(* Logix 5000 project; controller LeakTestAuto vendor 1 type 14 code 226 rev 37.11; software revision 37.01; part 2 of 13 *)
(* tags used below, declared in another part *)
   PLC : AOI_PLC;

ADD_ON_INSTRUCTION AOI_RFIDCompare   (* revision 1.0, ExecuteEnableInFalse *)
VAR_IN_OUT
   ExpectedResult : SINT[5,12]; {required}
   ExpectedResultIndex : DINT; {required}
END_VAR
VAR_OUTPUT
   Match : BOOL; {access Read Only, visible}
END_VAR
VAR_IN_OUT
   ReadBuffer : SINT[8000]; {required}
END_VAR
VAR
   i : DINT; {access None}
END_VAR

ROUTINE EnableInFalse   (* structured text *)
   Match := 0;
END_ROUTINE

ROUTINE Logic   (* structured text *)
   Match := 0;
   
   FOR i := 0 TO 11 DO
       IF ReadBuffer[i] <> ExpectedResult[ExpectedResultIndex, i] THEN
           EXIT;
       END_IF;
   END_FOR;
   
   IF i = 12 THEN
       Match := 1;
   END_IF;
END_ROUTINE
END_ADD_ON_INSTRUCTION

ADD_ON_INSTRUCTION AOI_RobotPositions   (* revision 1.0 *)
VAR_OUTPUT
   LoadingNest : DINT; {access Read Only}
   Barcode : DINT; {access Read Only}
   TestingNest1 : DINT; {access Read Only}
   TestingNest2 : DINT; {access Read Only}
   PassChute : DINT; {access Read Only}
   FailChute : DINT; {access Read Only}
END_VAR

ROUTINE Logic   (* structured text *)
   LoadingNest := 0;
   Barcode := 1;
   TestingNest1 := 2;
   TestingNest2 := 3;
   PassChute := 4;
   FailChute := 5;
END_ROUTINE
END_ADD_ON_INSTRUCTION

ADD_ON_INSTRUCTION AOI_Sequencer_x64   (* revision 1.0 *)
VAR_IN_OUT
   SequenceStructure : udt_SequenceStructure_X64; {required}
END_VAR
VAR_INPUT
   inpNextStepInterlock : BOOL; {access Read Only, required}
   inpCyclePause : BOOL; {access Read Only, required}
   inpStepMode : BOOL; {access Read Only, required}
END_VAR
VAR
   FFLUDumpREAL : REAL; {access None}
   Seq_FFLU_Cycle : CONTROL := (LEN := 10); {access None}
   Seq_FFLU_Step : CONTROL := (LEN := 64); {access None}
   Seq_FFLU_StepHist : CONTROL := (LEN := 64); {access None}
   FFLUDumpINT : INT; {access None}
   AvgContol : CONTROL := (LEN := 10); {access None}
END_VAR

ROUTINE Logic   (* ladder *)
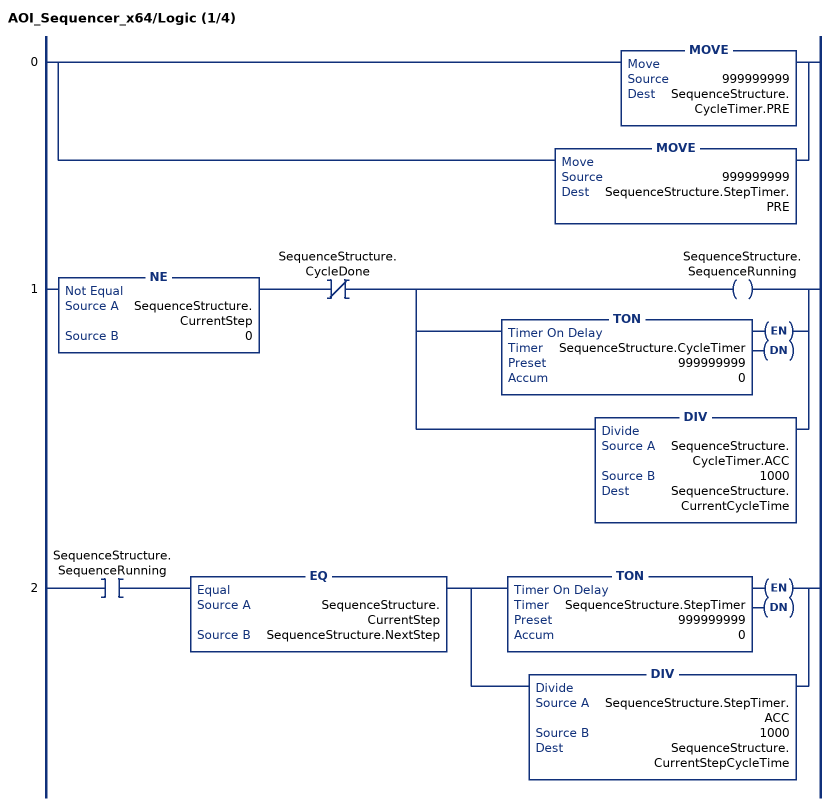
   0: [MOVE(999999999,SequenceStructure.CycleTimer.PRE) ,MOVE(999999999,SequenceStructure.StepTimer.PRE) ];
   1: NE(SequenceStructure.CurrentStep,0)XIO(SequenceStructure.CycleDone)[OTE(SequenceStructure.SequenceRunning) ,TON(SequenceStructure.CycleTimer,999999999,0) ,DIV(SequenceStructure.CycleTimer.ACC,1000,SequenceStructure.CurrentCycleTime) ];
   2: XIC(SequenceStructure.SequenceRunning)EQ(SequenceStructure.CurrentStep,SequenceStructure.NextStep)[TON(SequenceStructure.StepTimer,999999999,0) ,DIV(SequenceStructure.StepTimer.ACC,1000,SequenceStructure.CurrentStepCycleTime) ];
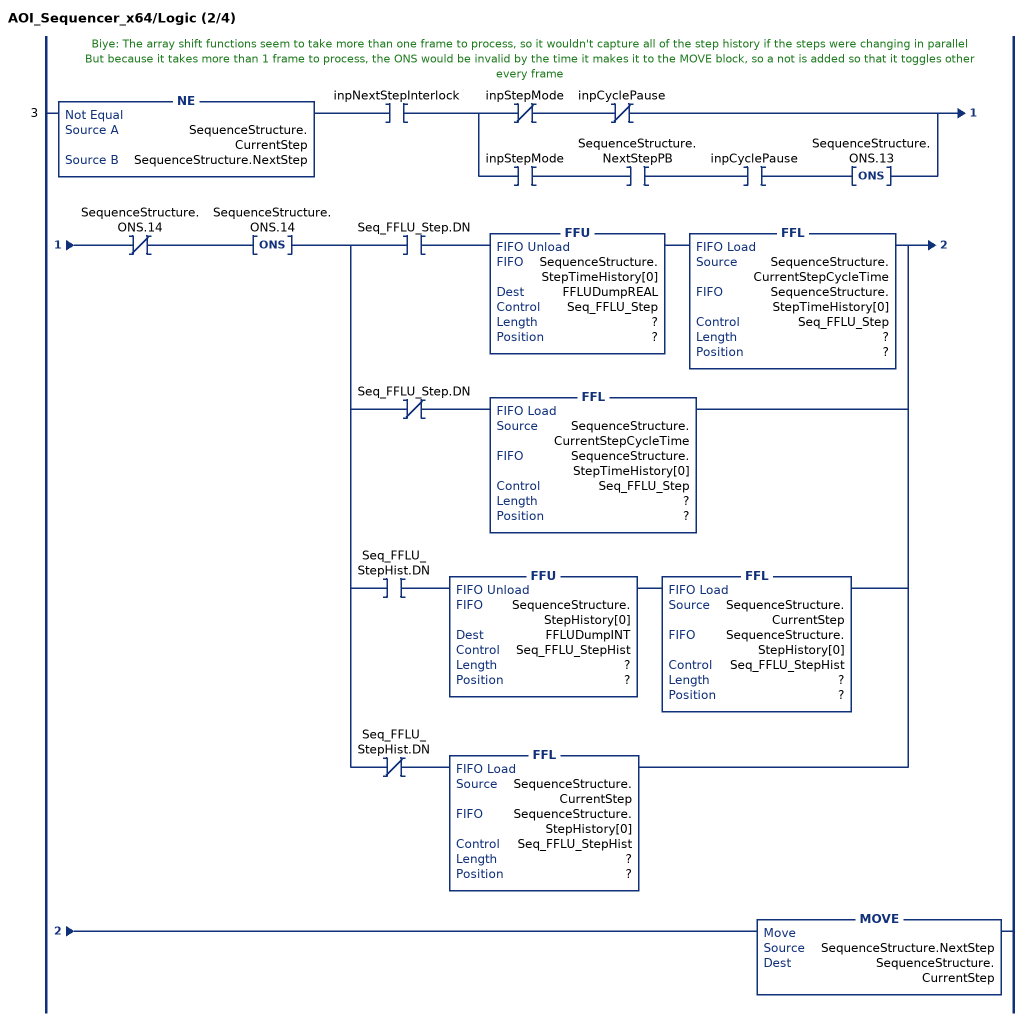
   // Biye: The array shift functions seem to take more than one frame to process, so it wouldn't capture all of the step history if the steps were changing in parallel
   // But because it takes more than 1 frame to process, the ONS would be invalid by the time it makes it to the MOVE block, so a not is added so that it toggles other every frame
   3: NE(SequenceStructure.CurrentStep,SequenceStructure.NextStep)XIC(inpNextStepInterlock)[XIO(inpStepMode) XIO(inpCyclePause) ,XIC(inpStepMode) XIC(SequenceStructure.NextStepPB) XIC(inpCyclePause) ONS(SequenceStructure.ONS.13) ]XIO(SequenceStructure.ONS.14)ONS(SequenceStructure.ONS.14)[XIC(Seq_FFLU_Step.DN) FFU(SequenceStructure.StepTimeHistory[0],FFLUDumpREAL,Seq_FFLU_Step,?,?) FFL(SequenceStructure.CurrentStepCycleTime,SequenceStructure.StepTimeHistory[0],Seq_FFLU_Step,?,?) ,XIO(Seq_FFLU_Step.DN) FFL(SequenceStructure.CurrentStepCycleTime,SequenceStructure.StepTimeHistory[0],Seq_FFLU_Step,?,?) ,XIC(Seq_FFLU_StepHist.DN) FFU(SequenceStructure.StepHistory[0],FFLUDumpINT,Seq_FFLU_StepHist,?,?) FFL(SequenceStructure.CurrentStep,SequenceStructure.StepHistory[0],Seq_FFLU_StepHist,?,?) ,XIO(Seq_FFLU_StepHist.DN) FFL(SequenceStructure.CurrentStep,SequenceStructure.StepHistory[0],Seq_FFLU_StepHist,?,?) ]MOVE(SequenceStructure.NextStep,SequenceStructure.CurrentStep);
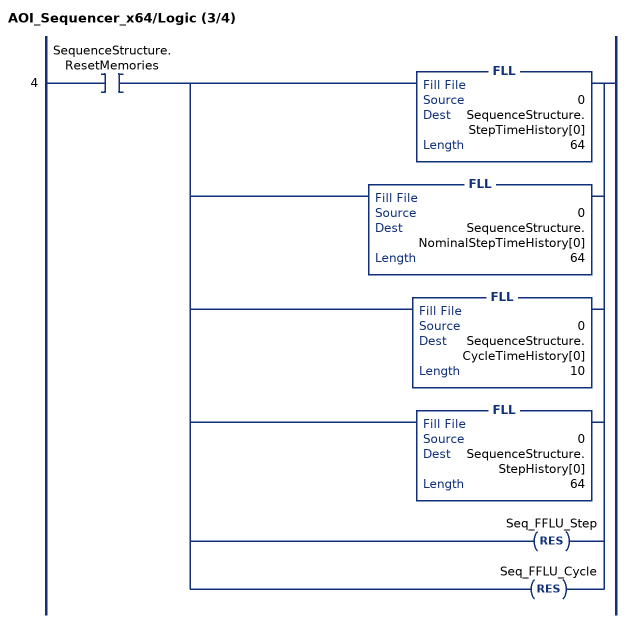
   4: XIC(SequenceStructure.ResetMemories)[FLL(0,SequenceStructure.StepTimeHistory[0],64) ,FLL(0,SequenceStructure.NominalStepTimeHistory[0],64) ,FLL(0,SequenceStructure.CycleTimeHistory[0],10) ,FLL(0,SequenceStructure.StepHistory[0],64) ,RES(Seq_FFLU_Step) ,RES(Seq_FFLU_Cycle) ];
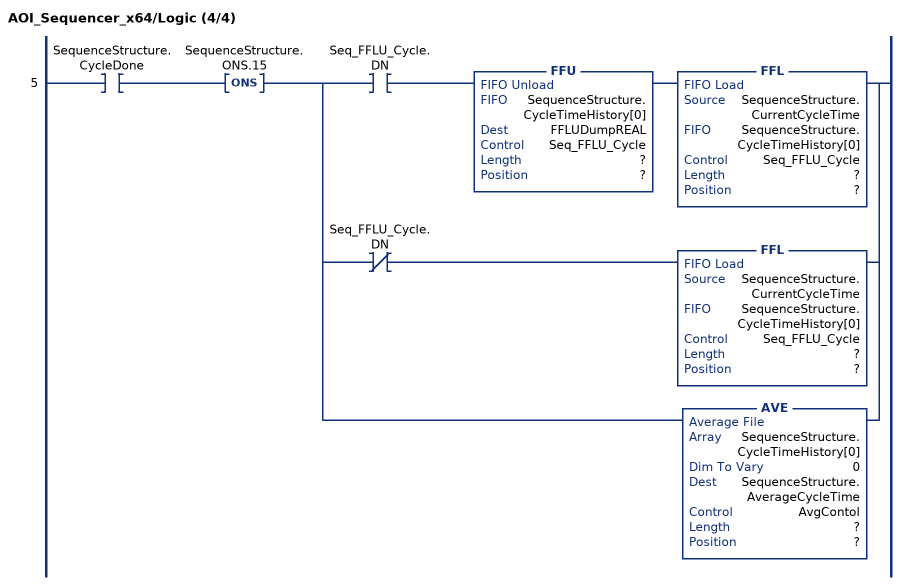
   5: XIC(SequenceStructure.CycleDone)ONS(SequenceStructure.ONS.15)[XIC(Seq_FFLU_Cycle.DN) FFU(SequenceStructure.CycleTimeHistory[0],FFLUDumpREAL,Seq_FFLU_Cycle,?,?) FFL(SequenceStructure.CurrentCycleTime,SequenceStructure.CycleTimeHistory[0],Seq_FFLU_Cycle,?,?) ,XIO(Seq_FFLU_Cycle.DN) FFL(SequenceStructure.CurrentCycleTime,SequenceStructure.CycleTimeHistory[0],Seq_FFLU_Cycle,?,?) ,AVE(SequenceStructure.CycleTimeHistory[0],0,SequenceStructure.AverageCycleTime,AvgContol,?,?) ];
END_ROUTINE
END_ADD_ON_INSTRUCTION

ADD_ON_INSTRUCTION AOI_StandardSeqSteps   (* revision 1.0 *)
VAR_OUTPUT
   Start : DINT; {access Read Only}
   ResultProcessing : DINT; {access Read Only}
   Complete : DINT; {access Read Only}
END_VAR

ROUTINE Logic   (* structured text *)
   Start := 1000;
   ResultProcessing := 8000;
   Complete := 9000;
END_ROUTINE
END_ADD_ON_INSTRUCTION

ADD_ON_INSTRUCTION INT_TO_BYTE   (* revision 1.0 *)
// It converts the INT to upper and lower nibbles
VAR_INPUT
   Input : INT;
END_VAR
VAR_OUTPUT
   OutUpperNibble : INT;
   OutLowerNibble : INT;
   iLowNib : INT; {access None}
   iUpNib : INT; {access None}
END_VAR

ROUTINE Logic   (* structured text *)
   iUpNib := Input/256;
   OutUpperNibble := iUpNib;
   iLowNib := Input -(iUpNib * 256);
   OutLowerNibble := iLowNib;
   
END_ROUTINE
END_ADD_ON_INSTRUCTION

ADD_ON_INSTRUCTION RWH_CMD   (* revision 1.1, ExecutePrescan *)
// AOI developed to handle to communicate with DTE102 , it handles 12 features of DTE 102.
// Revision note:
// Added isiModuleID, iiInputStartAdd, iiOutputStartAdd parameters for flexibility
VAR_IN_OUT
   iarsiInputFromDTE : SINT[496]; {required}   // Input array from DTE to PLC
END_VAR
VAR_INPUT
   ixConnOK : BOOL; {required}   // Connection to DTE from PLC, LIVE Status
   ixExecute : BOOL; {required}   // Rising edge : Execute selected user command.
   isiModuleID : SINT; {required}   // It indicates the module id set in the configuration to use each channel with different no of block size Please map this varible to DTE102:C.IO_x_module_identifier in controller tags. x = channel no on which RWH_CMD AOI is to be used
   iiInputStartAdd : INT; {required}   // It is the start of the DTE102:I from which the data has to be read depending upon the channel is being used by the user
   iiOutputStartAdd : INT; {required}   // It is the start of the DTE102:O to which the data has to be written depending upon the channel is being used by the user
   iiCmdCode : INT; {required}   // Command Mode for Function ID 11 and 12. For details refer user manual
   isiFunctionID : SINT; {required}   // ID of DTE10x command to be executed. For details refer user manual
   iiRdWrLength : INT; {required}   // data length (in BYTEs) to read/write USER memory on tag
   iiRdWrStartAddr : INT; {required}   // start address to read/write USER memory on tag
END_VAR
VAR_IN_OUT
   iarsiSendBuf : SINT[8000]; {required}   // send buffer for data to write to USER memory on tag
END_VAR
VAR_OUTPUT
   oxBusy : BOOL; {access Read Only, visible}   // Function block is busy, no new command possible
   oxDone : BOOL; {access Read Only, visible}   // TRUE: Operation resulted in error
   oxError : BOOL; {access Read Only, visible}   // TRUE: Operation resulted in error
   odiStatus : DINT; {access Read Only, visible}   // Status information or error code. For details refer user manual
   oxTagPresent : BOOL; {access Read Only, visible}   // TRUE : Tag present in field, FALSE : Tag not in field
   oiRcvdLength : INT; {access Read Only, visible}   // data length (in BYTEs) read from the tag
END_VAR
VAR_IN_OUT
   oarsiRcvBuf : SINT[8000]; {required}   // receive buffer for data from tag
END_VAR
VAR_OUTPUT
   oiDiagLength : INT; {access Read Only, visible}   // number of diagnostic data erros
END_VAR
VAR_IN_OUT
   oardiDiagData : DINT[4]; {required}   // Array with diagonostic data
   oarsiOutputToDTE : SINT[496]; {required}   // Output array from PLC to DTE
END_VAR
VAR
   iRcvdLength : INT;   // Local tag - calculates the received data length from PLC
   iLoopHandlerVar2 : INT;   // Local tag - Loop Handler variable 2
   iLoopHandlerVar1 : INT;   // Local tag - Loop Handler variable 1
   iActSizeOfSendBuf : INT;   // Local tag - Calculates the actual array size of the input array
   iActSizeOfRcvBuf : INT;   // Local tag - Calculates the actual array size of the recieve data array
   iActSizeOfOutputToDTE : INT;   // Local tag - Calculates the actual array size of the output array
   iActSizeOfInputFromDTE : INT;   // Local tag - Calculates the actual array size of the input array
   iBufferOffset : INT;   // Local tag - calculates the start adddress to read/write the data in buffer in case of ,ultiple cycles
   siActiveFunctionID : SINT;   // Loca tag - Latch the value of the selected ID to generate the error if t changes while function block is busy.
   siActiveModuleID : SINT; {access None}   // Local tag - indicates the active module id selected by user
   ciStateMachineSeparator : INT; {access None}   // Local tag = constant value of 1000. It separates the steps in state machine as per Function ID.
   iCmdCode : INT; {access None}   // Loca tag - Latch the value of the selected Cmd Code to generate the error if it changes while function block is busy.
   iLowerLimitInputStartAdd : INT; {access None}   // Local tag for limit the start address of input
   iUpperLimitInputStopAdderess : INT; {access None}   // Local tag - limit the upper range of input stop address
   iLowerLimitOutputStartAdd : INT; {access None}   // Local tag for limit the start address of output
   iUpperLimitOutputStopAdderess : INT; {access None}   // Local tag - limit the upper range of output stop address
   iActiveInputStartAdd : INT; {access None}   // Local Tag - Indicates the active input start adderess
   iActiveOutputStartAdd : INT; {access None}   // Local tag - Indicates the active output start address
   iArraySize : INT; {access None}
   iLengthToReadWriteInLastCycle : INT;   // Local tag to clculate the no of data byte to read/write in last cycle
   iNoCyclesReqToReadWriteCompleteData : INT;   // Local tag - Calculates the no of cycles required to read/write the data to/from DTE.
   iSingleCycleDataExchangeLimitInBytes : INT; {access None}   // Local tag - Decides the limit for bytes to exchange in one PLC cycle
   iTotalRcvdLength : INT; {access Read Only}   // data length (in BYTEs) read from the tag
   fb_OSRI_Execute : FBD_ONESHOT; {access None}   // Local tag - Detects the rising edge of the execute trigger. Avoids the multiple triggers for single command
   fb_DataAddress : INT_TO_BYTE; {access None}
   ardiDiagData : DINT[4]; {access None}   // Local tag -Array with diagonostic data
   xMultipleCyclesReq : BOOL;   // Local tag - Status for single or multiple cycle requirement to read / write data. if xMultipleCyclesReq = 0 then data transmission takes one cycle else it takes >1 cycles.
   fb_CmdCode : INT_TO_BYTE; {access None}   // Local tag = function block to convert cmd code to MSB and LSB.
   fb_OSRI_TagPresent : FBD_ONESHOT; {access None}   // Local tag = checks for tag present rising edge to read / write asynchronous commands
   fb_DataLength : INT_TO_BYTE; {access None}
   fb_SINT_TO_INT : SINT_TO_INT; {access None}
   scDTE102_Handling : DTE102_CmdModule; {access None}
   iStateMachine_RWH_CMD : INT;   // Local tag - State machine handling variable for AOI logic
END_VAR

ROUTINE Logic   (* structured text *)
   (*// ******************************************************************************************************
   // Disclaimer OF Warranties
   (*
   	ifm disclaims to the fullest extent authorized by law any and all warranties,
   	whether express or implied, including, without limitation,
   	any implied warranties of title, non-infringement, quiet enjoyment,
   	integration, merchantability or fitness for a particular purpose.
   
   	Without limitation of the foregoing, ifm expressly does not warrant that:
   	(a)  the software will meet your requirements or expectations;
   	(b)  the software or the software content will be free of bugs, errors,
   			 viruses or other defects;
   	(c)  any results, output, or data provided through or generated by the software
   			 will be accurate, up-to-date, complete or reliable;
   	(d)  the software will be compatible with third party software;
   	(e)  any errors in the software will be corrected
   
   
   	DEMO SOFTWARE AND TEMPLATES
   
   	Demo software and templates are provided “as is” and “as available”,
   	without any warranty of any kind, either express or implied.
   	The User acknowledges and agrees to use the software at User’s own risk.
   	In no event shall ifm be held liable for any direct, indirect, incidental
   	or consequential damages arising out of the use of or inability to use the software.
   	User may use the software solely for demonstration purposes
   	and to assess the software functionalities and capabilities.
   
   
   	Software written specifically for Customer
   
   	1. The software created and used is put together by ifm specially to the customer
   		 using modular software components made by ifm for numerous applications (Standard software modules)
   		 and adapted to the contractual service required (customer-specific application program).
   
   	2. Upon complete payment of the purchase price for the customer-specific application program,
   		 ifm transfers the non-exclusive, locally and temporarily unrestricted usage right
   		 thereof to the customer, without the customer acquiring any rights of any kind
   		 to the standard software module on which the individual or customer-specific adaptation is based.
   		 Notwithstanding these provisions, ifm reserves the right to produce and offer
   		 customer specific software solutions of the same kind for other customers
   		 based on other terms of reference. In any case ifm retains a simple right of usage
   		 of the customer–specific solution for internal purposes.
   
   	3. Upon acceptance of the program, User acknowledges and agrees to use the software
   		 at User’s own risk. User also acknowledges and agrees upon acceptance of the program
   		 that the software meets the requirements of the specifications agreed upon.
   		 ifm disclaims any and all warranties, in particular regarding fitness of the software
   		 for a particular purpose.
   ******************************************************************************************************
   *)
   (* Revision history:
   3rd June 2022:
   New Chnage requests:
   1. check if the "get diagdata" command is send if TP bit is high and no command active
      DiagData before sending a command --> get Diagnostic shall be send automatically before executing a user command.
   
   
   24th Dec 2020:
   Fixed bug:
   	Whenever customer tries to read (one time) from offset=10, length = 10 bytes, the data is read from offset=0
   	Same for writing (one time) and write verifed (one time) operations too.
   
   26th July 2019:
   	Till now, it was assumed that after diagnostic read, maximum number of reported errors could be 4 only.
   	But, actually errors are to be read, until DIAG bit is active.
   	Fixed this in the code.
   
   19th July 2019:
   	Added following check.
   	When a execute trigger is given, and already some operation is in progress (TA <> TR).
   	Now, we wait for ongoing operation to complete.
   
   17th July 2019:
   	i. Write-verified operation: Added extra check, that the number of recieved bytes should be same as requested "iiRdWrLength"
   	ii. Added a logic to report error, in case device reports error and provides no error codes.
   
   16th July 2019:
   	i. Fixed following bugs:
   	All 4 channels were used, and given a command of "write verified" one time.
   	For every alternate channel, operation resulted in error.
   	Reason: While waiting for user action, the TR bit was not maintained same as TA
   
   9th July 2019
   	Fixed following bugs:
   	i. Parallel usage of all 4 channels, with configuration 17,17,17,14 was buggy.
   	Reason: Every fb instance's trigger reset, was overwritting DTE fieldbus output array.
   
   	ii. Write verfied was not working for channel, with module id 12. RdWrLength = 8000 bytes
   	Reason: The number of bytes to be written in last cyle, was not calculated correctly.
   *)
   (*
   Status codes:
   	0x0000 	Function completed without error.
   	0x1000	Waiting for ixConnOk = TRUE, input parameter
   	0x7000	Wait for start of command
   	0x7001	Wait for Rising edge of the TP Bit in case of asynchronous commands
   	0x7102	Read the USER Memory
   	0x7103	Complete reading of the USER Memory
   	0x7202	Write to the USER Memory
   	0x7203	Complete writing to the USER Memory
   	0x7302	Read UID
   	0x7303	Complete reading UID
   	0x7402	Read Diagnostic data
   	0x7403	Complete reading the Diagnostic data
   	0x7501	Antenna OFF command
   	0x7502	Complete Antenna OFF command
   	0x7601	Antenna ON command
   	0x7602	Complete Antenna ON command
   	0x7701	Read device parameters one time Command
   	0x7702	Complete read device parameters one time command
   	0x7801	Set device parameters one time Command
   	0x7802	Complete Set device parameters one time command
   
   Error codes:
   	0x8000 	Evaluation unit indicates an error; evaluate the diagnostic data in the oardiDiagData output parameter. For the error codes see the device manual
   	0x8101 	isiFunctionID input parameter invalid
   
   	0x8104	Different sizes of the iarsiInputFromDTE input parameter and oarsiOutputToDTE output parameter
   	0x8107	iiCmdCode = Invalid, but selected ID is 11 or 12
   	0x8109	iiRdWrStartAddr input is invalid
   	0x8110	Antenna already OFF.
   	0x8111	Antenna already ON.
   	0x8112	Wrong Module ID entered by user
   	0x8113	Wrong Input Start Address entered by user
   	0x8114	Wrong Output Start Address entered by user
   	0x8201	ixConnOk input parameter = FALSE during command execution.
   	0x8301	Start of a command while the function block is busy (oxBusy = TRUE)
   	0x8302	Start of a command with antenna switched off.
   	0x8303	Function ID changed while function block is BUSY.
   	0x8304	Start of a command without tag in the antenna field
   	0x8305	iiRdWrLength input parameter <= 0 or greater than the defined receive buffer (oarsiRcvBuf)
   	0x8306	iiRdWrLength input parameter <= 0 or greater than the defined send buffer (iarsiSendBuf)
   	0x8307	Invalid Read Write data length if asynchronous command is selected
   	0x8308	Command Code changed while function block is BUSY.
   	0x8309	Module ID changed when function block is BUSY
   	0x8310	Input start address changed when function block is BUSY
   	0x8311	Output start address changed when function block is BUSY
   	0x8313 	Write-verified: Complete data could not be written
   	0x8314  Device reported error, but provided no diagonostic codes
    	0x8315	Read data: Complete data could not be read
   	0x8316	Write data: Complete data could not be written
   *)
   	// Execute Trigger
   	fb_OSRI_Execute.InputBit := ixExecute;
   	OSRI(fb_OSRI_Execute);
   
   	// If function block is busy and following conditions occure then go to error state
   	// 1. Connection Lost
   	// 2. Multiple Execute Triggers
   	// 3. ID Change by user
   	// 4. Command code changed by the user
   	// 5. Module ID changed by the user
   	// 6. Input start add changed by the user
   	// 7. Output start add changed by the user
   
   	IF(iStateMachine_RWH_CMD > 0 AND iStateMachine_RWH_CMD < 20000)THEN
   		IF(NOT(ixConnOK))THEN							// No Connection to DTE
   			oxBusy := 1;
   			oxDone := 0;
   			oxError := 0;
   			odiStatus := 16#8201; //ixConnOk input parameter = FALSE during command execution.
   			iStateMachine_RWH_CMD := 20000;
   		ELSIF(fb_OSRI_Execute.OutputBit)THEN			// Multiple Execute Triggers
   			oxBusy := 1;
   			oxDone := 0;
   			oxError := 0;
   			odiStatus := 16#8301; //Start of a command while the function block is busy (oxBusy = TRUE)
   			iStateMachine_RWH_CMD := 20000;
   		ELSIF(isiFunctionID<>siActiveFunctionID)THEN	// Function ID Changed by user when function is Active
   			oxBusy := 1;
   			oxDone := 0;
   			oxError := 0;
   			odiStatus := 16#8303; //Function ID changed while function block is BUSY.
   			iStateMachine_RWH_CMD := 20000;
   		ELSIF(iiCmdCode <> iCmdCode)THEN				// Command code changed by user when function is Active
   			oxBusy := 1;
   			oxDone := 0;
   			oxError := 0;
   			odiStatus := 16#8308; //Command Code changed while function block is BUSY.
   			iStateMachine_RWH_CMD := 20000;
   		ELSIF(siActiveModuleID <> isiModuleID)THEN
   			oxBusy := 1;
   			oxDone := 0;
   			oxError := 0;
   			odiStatus := 16#8309; 						// Module ID changed by user when function is Active
   			iStateMachine_RWH_CMD := 20000;
   		ELSIF(iActiveInputStartAdd <> iiInputStartAdd)THEN
   			oxBusy := 1;
   			oxDone := 0;
   			oxError := 0;
   			odiStatus := 16#8310; 						// Input Start Address changed by user when function is Active
   			iStateMachine_RWH_CMD := 20000;
   		ELSIF(iActiveOutputStartAdd <> iiOutputStartAdd)THEN
   			oxBusy := 1;
   			oxDone := 0;
   			oxError := 0;
   			odiStatus := 16#8311; 						// Output Start Address changed by user when function is Active
   			iStateMachine_RWH_CMD := 20000;
   		END_IF;
   	END_IF;
   
   	IF(iiInputStartAdd >= 0 AND iiInputStartAdd < 496)AND(iiOutputStartAdd >= 0 AND iiOutputStartAdd < 496)THEN
   		// Maping of Input bits
   		scDTE102_Handling.Status.TP		:=	iarsiInputFromDTE[iiInputStartAdd].0;
   		scDTE102_Handling.Status.AI 	:=	iarsiInputFromDTE[iiInputStartAdd].1;
   		scDTE102_Handling.Status.WA 	:=	iarsiInputFromDTE[iiInputStartAdd].2;
   		scDTE102_Handling.Status.RA 	:=	iarsiInputFromDTE[iiInputStartAdd].3;
   		scDTE102_Handling.Status.UA 	:=	iarsiInputFromDTE[iiInputStartAdd].4;
   		scDTE102_Handling.Status.EA 	:=	iarsiInputFromDTE[iiInputStartAdd].5;
   		scDTE102_Handling.Status.DA 	:=	iarsiInputFromDTE[iiInputStartAdd].6;
   		scDTE102_Handling.Status.DIAG	:=	iarsiInputFromDTE[iiInputStartAdd].7;
   
   
   		scDTE102_Handling.Status.TA						:=	iarsiInputFromDTE[iiInputStartAdd+1].0;
   		iarsiInputFromDTE[iiInputStartAdd+1].1			:=	iarsiInputFromDTE[iiInputStartAdd+1].1;
   		iarsiInputFromDTE[iiInputStartAdd+1].2 			:=	iarsiInputFromDTE[iiInputStartAdd+1].2;
   		iarsiInputFromDTE[iiInputStartAdd+1].3 			:=	iarsiInputFromDTE[iiInputStartAdd+1].3;
   		iarsiInputFromDTE[iiInputStartAdd+1].4 			:=	iarsiInputFromDTE[iiInputStartAdd+1].4;
   		iarsiInputFromDTE[iiInputStartAdd+1].5 			:=	iarsiInputFromDTE[iiInputStartAdd+1].5;
   		iarsiInputFromDTE[iiInputStartAdd+1].6 			:=	iarsiInputFromDTE[iiInputStartAdd+1].6;
   		scDTE102_Handling.Status.CA 					:=	iarsiInputFromDTE[iiInputStartAdd+1].7;
   	END_IF;
   
   	// Mapping tag Present bit to output variable
   	oxTagPresent := scDTE102_Handling.Status.TP;
   
   	// Asynchronous commands :- Check For tag Present bit
   	fb_OSRI_TagPresent.InputBit := scDTE102_Handling.Status.TP;
   	OSRI(fb_OSRI_TagPresent);
   
   
   CASE iStateMachine_RWH_CMD OF
   	/// This case checks the inputs entered by user properly or not.
   	0:
   		scDTE102_Handling.ActivateCommand.TR	:= (iarsiInputFromDTE[iiInputStartAdd+1].0); //Do not accidently trigger a command
   
   		// getting the sizes of arrays used in function block to check correct sizes declared by user.
   		SIZE(iarsiInputFromDTE,0,iActSizeOfInputFromDTE);
   		SIZE(oarsiOutputToDTE,0,iActSizeOfOutputToDTE);
   		SIZE(iarsiSendBuf,0,iActSizeOfSendBuf);
   		SIZE(oarsiRcvBuf,0,iActSizeOfRcvBuf);
   
   		// Logic to identify the module ID and related Data buffer size required for operations and start address for reading and writting
   		CASE isiModuleID OF
   			12 :
   				iLowerLimitInputStartAdd := 0;
   				iUpperLimitInputStopAdderess := iActSizeOfInputFromDTE - 26;
   				iLowerLimitOutputStartAdd := 0;
   				iUpperLimitOutputStopAdderess := iActSizeOfOutputToDTE - 26;
   				iSingleCycleDataExchangeLimitInBytes := 20;
   			13 :
   				iLowerLimitInputStartAdd := 0;
   				iUpperLimitInputStopAdderess := iActSizeOfInputFromDTE - 46;
   				iLowerLimitOutputStartAdd := 0;
   				iUpperLimitOutputStopAdderess := iActSizeOfOutputToDTE - 46;
   				iSingleCycleDataExchangeLimitInBytes := 40;
   			14 :
   				iLowerLimitInputStartAdd := 0;
   				iUpperLimitInputStopAdderess := iActSizeOfInputFromDTE - 66;
   				iLowerLimitOutputStartAdd := 0;
   				iUpperLimitOutputStopAdderess := iActSizeOfOutputToDTE - 66;
   				iSingleCycleDataExchangeLimitInBytes := 60;
   			15 :
   				iLowerLimitInputStartAdd := 0;
   				iUpperLimitInputStopAdderess := iActSizeOfInputFromDTE - 86;
   				iLowerLimitOutputStartAdd := 0;
   				iUpperLimitOutputStopAdderess := iActSizeOfOutputToDTE - 86;
   				iSingleCycleDataExchangeLimitInBytes := 80;
   			16 :
   				iLowerLimitInputStartAdd := 0;
   				iUpperLimitInputStopAdderess := iActSizeOfInputFromDTE - 106;
   				iLowerLimitOutputStartAdd := 0;
   				iUpperLimitOutputStopAdderess := iActSizeOfOutputToDTE - 106;
   				iSingleCycleDataExchangeLimitInBytes := 100;
   			17 :
   				iLowerLimitInputStartAdd := 0;
   				iUpperLimitInputStopAdderess := iActSizeOfInputFromDTE - 126;
   				iLowerLimitOutputStartAdd := 0;
   				iUpperLimitOutputStopAdderess := iActSizeOfOutputToDTE - 126;
   				iSingleCycleDataExchangeLimitInBytes := 120;
   			18 :
   				iLowerLimitInputStartAdd := 0;
   				iUpperLimitInputStopAdderess := iActSizeOfInputFromDTE - 146;
   				iLowerLimitOutputStartAdd := 0;
   				iUpperLimitOutputStopAdderess := iActSizeOfOutputToDTE - 146;
   				iSingleCycleDataExchangeLimitInBytes := 140;
   			19 :
   				iLowerLimitInputStartAdd := 0;
   				iUpperLimitInputStopAdderess := iActSizeOfInputFromDTE - 166;
   				iLowerLimitOutputStartAdd := 0;
   				iUpperLimitOutputStopAdderess := iActSizeOfOutputToDTE - 166;
   				iSingleCycleDataExchangeLimitInBytes := 160;
   		END_CASE;
   
   		// Checking all input parameters
   		IF(fb_OSRI_Execute.OutputBit)THEN //Received trigger
   			oxBusy := 1;
   			oxDone := 0;
   			oxError := 0;
   			IF(NOT(ixConnOK))THEN
   				odiStatus := 16#8201;					// ixConnOk input parameter = FALSE during command execution.
   				iStateMachine_RWH_CMD := 20000;
   			ELSIF(isiModuleID < 12 OR isiModuleID > 19)THEN
   				odiStatus := 16#8112;					// Wrong Module ID entered by user.
   				iStateMachine_RWH_CMD := 20000;
   			ELSIF(iiInputStartAdd < iLowerLimitInputStartAdd OR iiInputStartAdd > iUpperLimitInputStopAdderess)THEN
   				odiStatus := 16#8113;					// Wrong Input Start Address entered by user.
   				iStateMachine_RWH_CMD := 20000;
   			ELSIF(iiOutputStartAdd < iLowerLimitOutputStartAdd OR iiOutputStartAdd > iUpperLimitOutputStopAdderess)THEN
   				odiStatus := 16#8114;					// Wrong Output Start Address entered by user.
   				iStateMachine_RWH_CMD := 20000;
   			ELSIF(isiFunctionID < 1 OR isiFunctionID > 12)THEN
   				odiStatus := 16#8101;					// isiFunctionID input parameter invalid
   				iStateMachine_RWH_CMD := 20000;
   			ELSIF((isiFunctionID = 11 AND(iiCmdCode<>25288 AND iiCmdCode<>25289 AND (iiCmdCode < 25293 OR iiCmdCode > 25299))) OR
   			  	 (isiFunctionID = 12 AND (iiCmdCode< 26070 OR iiCmdCode > 26077)))THEN
   				odiStatus := 16#8107;					// iiCmdCode = Invalid, but selected ID is 11 or 12
   				iStateMachine_RWH_CMD := 20000;
   			ELSIF(iActSizeOfInputFromDTE <> iActSizeOfOutputToDTE)THEN
   				odiStatus := 16#8104;					// Different sizes of the iarsiInputFromDTE input parameter and oarsiOutputToDTE output parameter
   				iStateMachine_RWH_CMD := 20000;
   			ELSIF((iiRdWrLength < 1 or iiRdWrLength > iActSizeOfRcvBuf)AND(isiFunctionID <> 9 AND isiFunctionID <> 10 AND isiFunctionID <> 1 AND isiFunctionID <> 2 AND isiFunctionID <> 11 AND isiFunctionID <> 12)) OR
   				 ((iiRdWrLength < 1 or iiRdWrLength > iActSizeOfRcvBuf) AND((isiFunctionID = 11 AND iiCmdCode = 16#62D1)OR(isiFunctionID = 12 AND iiCmdCode = 16#65D8)))THEN
   				odiStatus := 16#8305;					// iiRdWrLength input parameter <= 0 or greater than the defined receive buffer (oarsiRcvBuf)
   				iStateMachine_RWH_CMD := 20000;
   			ELSIF((iiRdWrLength < 1 or iiRdWrLength > iActSizeOfSendBuf)AND(isiFunctionID <> 9 AND isiFunctionID <> 10 AND isiFunctionID <> 1 AND isiFunctionID <> 2 AND isiFunctionID <> 11 AND isiFunctionID <> 12)) OR
   				 ((iiRdWrLength < 1 or iiRdWrLength > iActSizeOfSendBuf) AND((isiFunctionID = 11 AND iiCmdCode = 16#62D1)OR(isiFunctionID = 12 AND iiCmdCode = 16#65D8)))THEN
   				odiStatus := 16#8306;					// iiRdWrLength input parameter <= 0 or greater than the defined send buffer (iarsiSendBuf)
   				iStateMachine_RWH_CMD := 20000;
   			ELSIF(iiRdWrLength < 1 or iiRdWrLength > (iSingleCycleDataExchangeLimitInBytes))AND((isiFunctionID = 3)OR(isiFunctionID = 5)OR(isiFunctionID = 7))THEN
   				odiStatus := 16#8307;					// Invalid Read Write data length if asynchronous command is selected.
   				iStateMachine_RWH_CMD := 20000;
   			ELSIF(scDTE102_Handling.Status.AI)AND(isiFunctionID <> 9)AND(isiFunctionID <> 10)THEN
   				odiStatus := 16#8302;					// Start of a command with antenna switched off.
   				iStateMachine_RWH_CMD := 20000;
   			ELSIF(NOT(oxTagPresent))AND(isiFunctionID <> 9)AND(isiFunctionID <> 10)AND(isiFunctionID <> 3)AND(isiFunctionID <> 5)AND(isiFunctionID <> 7)AND(isiFunctionID <> 1)THEN
   				odiStatus := 16#8304;					// Start of a command without tag in the antenna field
   				iStateMachine_RWH_CMD := 20000;
   			ELSIF((iiRdWrStartAddr < 0 OR iiRdWrStartAddr > (iActSizeOfSendBuf-iiRdWrLength))AND(isiFunctionID <> 9 AND isiFunctionID <> 10 AND isiFunctionID <> 1 AND isiFunctionID <> 2 AND isiFunctionID <> 11 AND isiFunctionID <> 12)) OR
   				 ((iiRdWrStartAddr < 0 OR iiRdWrStartAddr > (iActSizeOfSendBuf-iiRdWrLength)) AND((isiFunctionID = 11 AND iiCmdCode = 16#62D1)OR(isiFunctionID = 12 AND iiCmdCode = 16#65D8)))THEN
   				odiStatus := 16#8109;					// iiRdWrStartAddr input is invalid
   				iStateMachine_RWH_CMD := 20000;
   			ELSIF(isiFunctionID = 9)AND(scDTE102_Handling.Status.AI)THEN
   				odiStatus := 16#8110;					// Antenna already OFF.
   				iStateMachine_RWH_CMD := 20000;
   			ELSIF(isiFunctionID = 10)AND(NOT(scDTE102_Handling.Status.AI))THEN
   				odiStatus := 16#8111;					// Antenna already ON.
   				iStateMachine_RWH_CMD := 20000;
   			ELSE
   				siActiveFunctionID := isiFunctionID;	// All input parameters are valid. Start executing the selected ID.
   				iCmdCode := iiCmdCode;
   				ciStateMachineSeparator := 1000;		//cStateMachineSeparator := 1000;
   				siActiveModuleID := isiModuleID;
   				iActiveInputStartAdd := iiInputStartAdd;
   				iActiveOutputStartAdd := iiOutputStartAdd;
   				iStateMachine_RWH_CMD := 7110;
   
   			END_IF;
   		ELSE //no trigger recieved yet
   			IF(NOT(ixConnOK))THEN
   				oxBusy := 0;
   				oxDone := 0;
   				oxError := 0;
   				odiStatus := 16#1000;					//No connection to DTE.
   				iStateMachine_RWH_CMD := 0;
   			ELSE
   				oxBusy := 0;
   				oxDone := 0;
   				oxError := 0;
   				odiStatus := 16#7000;					// Connection OK, Waiting for Command.
   				iStateMachine_RWH_CMD := 0;
   			END_IF;
   		END_IF;
   
   // Get automatically existing diagnostic data before executing new user command.
   
   	7110:
   		IF(scDTE102_Handling.Status.DIAG)THEN		//  Existing Error is present
   			oxBusy := 1;
   			oxDone := 0;
   			oxError := 0;
   			scDTE102_Handling.ActivateCommand.AO	:= 0;
   			scDTE102_Handling.ActivateCommand.WR	:= 0;
   			scDTE102_Handling.ActivateCommand.RD	:= 0;
   			scDTE102_Handling.ActivateCommand.UR	:= 0;
   			scDTE102_Handling.ActivateCommand.ER	:= 0;
   			scDTE102_Handling.ActivateCommand.DR	:= 1;
   			scDTE102_Handling.ActivateCommand.CM	:= 0;
   			scDTE102_Handling.ActivateCommand.TR	:= NOT(scDTE102_Handling.Status.TA);
   			odiStatus := 16#7402;
   			iStateMachine_RWH_CMD					:= 7111;
   		ELSIF NOT(scDTE102_Handling.Status.TA XOR scDTE102_Handling.ActivateCommand.TR)THEN // Proceed,when TA=TR
   			iStateMachine_RWH_CMD := siActiveFunctionID * ciStateMachineSeparator;
   		END_IF;
   
   	7111:// waiting for fieldbus to free
   		IF NOT(scDTE102_Handling.Status.TA XOR scDTE102_Handling.ActivateCommand.TR)THEN // Proceed,when TA=TR
   			iStateMachine_RWH_CMD					:= 7112;
   		end_if;
   
   	7112:
   		IF (scDTE102_Handling.Status.DIAG)THEN		//   IF Error is present
   			oxBusy := 1;
   			oxDone := 0;
   			oxError := 0;
   			scDTE102_Handling.ActivateCommand.AO	:= 0;
   			scDTE102_Handling.ActivateCommand.WR	:= 0;
   			scDTE102_Handling.ActivateCommand.RD	:= 0;
   			scDTE102_Handling.ActivateCommand.UR	:= 0;
   			scDTE102_Handling.ActivateCommand.ER	:= 0;
   			scDTE102_Handling.ActivateCommand.DR	:= 1;
   			scDTE102_Handling.ActivateCommand.CM	:= 0;
   			scDTE102_Handling.ActivateCommand.TR	:= NOT(scDTE102_Handling.Status.TA);
   			odiStatus := 16#7402;
   			iStateMachine_RWH_CMD					:= 19000;
   		ELSIF NOT(scDTE102_Handling.Status.TA XOR scDTE102_Handling.ActivateCommand.TR)THEN // Proceed,when TA=TR
   			iStateMachine_RWH_CMD := siActiveFunctionID * ciStateMachineSeparator;
   		END_IF;
   
   	// Function ID 1 :- read the UID of the ID-tag continuously
   	1000:
   		// frame a command and send to the DTE.
   		scDTE102_Handling.ActivateCommand.AO	:= 0;
   		scDTE102_Handling.ActivateCommand.WR	:= 0;
   		scDTE102_Handling.ActivateCommand.RD	:= 0;
   		scDTE102_Handling.ActivateCommand.UR	:= 0;
   		scDTE102_Handling.ActivateCommand.ER	:= 0;
   		scDTE102_Handling.ActivateCommand.DR	:= 0;
   		scDTE102_Handling.ActivateCommand.CM	:= 0;
   		oarsiOutputToDTE[iiOutputStartAdd+2]	:= 0;
   		oarsiOutputToDTE[iiOutputStartAdd+3]	:= 0;
   		oarsiOutputToDTE[iiOutputStartAdd+4]	:= 0;
   		oarsiOutputToDTE[iiOutputStartAdd+5]	:= 0;
   		scDTE102_Handling.ActivateCommand.TR	:= NOT(scDTE102_Handling.Status.TA);
   		odiStatus := 16#7302;
   		iStateMachine_RWH_CMD					:= 1050;
   
   
   	1050:
   		IF(scDTE102_Handling.Status.DIAG)THEN		// Error in receiving  the data from DTE.
   			oxBusy := 1;
   			oxDone := 0;
   			oxError := 0;
   			scDTE102_Handling.ActivateCommand.AO	:= 0;
   			scDTE102_Handling.ActivateCommand.WR	:= 0;
   			scDTE102_Handling.ActivateCommand.RD	:= 0;
   			scDTE102_Handling.ActivateCommand.UR	:= 0;
   			scDTE102_Handling.ActivateCommand.ER	:= 0;
   			scDTE102_Handling.ActivateCommand.DR	:= 1;
   			scDTE102_Handling.ActivateCommand.CM	:= 0;
   			oarsiOutputToDTE[iiOutputStartAdd+2]	:= 16#00;
   			scDTE102_Handling.ActivateCommand.TR	:= NOT(scDTE102_Handling.Status.TA);
   			odiStatus := 16#7402;
   			iStateMachine_RWH_CMD					:= 19000;
   		ELSE										// ElSE condition, no error then read the status from the DTE.
   			IF(NOT(scDTE102_Handling.Status.TA XOR scDTE102_Handling.ActivateCommand.TR))THEN // Proceed,when TA=TR
   				SINT_TO_INT(fb_SINT_TO_INT,iarsiInputFromDTE[iiInputStartAdd+3]);
   				iRcvdLength := fb_SINT_TO_INT.oINT_var;
   				IF(iRcvdLength <> 0)THEN //Data read is non zero
   					oiRcvdLength := (iRcvdLength-2);			// Subtract 2 from actual length which is RSSI length.
   					CPS(iarsiInputFromDTE[iiInputStartAdd+6],oarsiRcvBuf[0],oiRcvdLength);
   					odiStatus := 16#7303;
   					iStateMachine_RWH_CMD := 13000;
   				ELSIF(NOT(scDTE102_Handling.Status.TP))THEN
   					oxBusy := 1;
   					oxDone := 0;
   					oxError := 0;
   					odiStatus := 16#7001;
   					iStateMachine_RWH_CMD := 1050;
   				END_IF;
   			END_IF;
   		END_IF;
   
   	// Function ID 2 :- read the UID of the ID-tag one time
   	2000:
   		// frame a command and send to the DTE.
   		scDTE102_Handling.ActivateCommand.AO	:= 0;
   		scDTE102_Handling.ActivateCommand.WR	:= 0;
   		scDTE102_Handling.ActivateCommand.RD	:= 1;
   		scDTE102_Handling.ActivateCommand.UR	:= 0;
   		scDTE102_Handling.ActivateCommand.ER	:= 0;
   		scDTE102_Handling.ActivateCommand.DR	:= 0;
   		scDTE102_Handling.ActivateCommand.CM	:= 1;
   		oarsiOutputToDTE[iiOutputStartAdd+2]	:= 0;
   		oarsiOutputToDTE[iiOutputStartAdd+3]	:= 16#02;
   		oarsiOutputToDTE[iiOutputStartAdd+4]	:= 16#62;
   		oarsiOutputToDTE[iiOutputStartAdd+5]	:= 16#CD;
   		scDTE102_Handling.ActivateCommand.TR	:= NOT(scDTE102_Handling.Status.TA);
   		odiStatus := 16#7302;
   		iStateMachine_RWH_CMD					:= 2050;
   
   
   	2050:
   		IF(scDTE102_Handling.Status.DIAG)THEN		// Error in receiving  the data from DTE.
   			oxBusy := 1;
   			oxDone := 0;
   			oxError := 0;
   			scDTE102_Handling.ActivateCommand.AO	:= 0;
   			scDTE102_Handling.ActivateCommand.WR	:= 0;
   			scDTE102_Handling.ActivateCommand.RD	:= 0;
   			scDTE102_Handling.ActivateCommand.UR	:= 0;
   			scDTE102_Handling.ActivateCommand.ER	:= 0;
   			scDTE102_Handling.ActivateCommand.DR	:= 1;
   			scDTE102_Handling.ActivateCommand.CM	:= 0;
   			oarsiOutputToDTE[iiOutputStartAdd+2]	:= 16#00;
   			scDTE102_Handling.ActivateCommand.TR	:= NOT(scDTE102_Handling.Status.TA);
   			odiStatus := 16#7402;
   			iStateMachine_RWH_CMD					:= 19000;
   		ELSE										// ElSE condition, no error then read the status from the DTE.
   			IF(NOT(scDTE102_Handling.Status.TA XOR scDTE102_Handling.ActivateCommand.TR))AND(scDTE102_Handling.Status.CA)THEN
   				oiRcvdLength := (iarsiInputFromDTE[iiInputStartAdd+7]-2);			// Subtract 2 from actual length which is RSSI length.
   				CPS(iarsiInputFromDTE[iiInputStartAdd+10],oarsiRcvBuf[0],oiRcvdLength);
   				odiStatus := 16#7303;
   				iStateMachine_RWH_CMD := 18000;
   			END_IF;
   		END_IF;
   
   
   	// Function ID 3 :- read an area of the USER memory of the ID-tag automatically
   	3000:
   		// frame a command and send to the DTE.
   		IF(iiRdWrLength <= (iSingleCycleDataExchangeLimitInBytes))THEN	// User memory can be read in single cycle
   			xMultipleCyclesReq  := 0;
   			fb_DataLength.Input := iiRdWrLength;
   			fb_DataAddress.Input:= iiRdWrStartAddr;
   			odiStatus := 16#7102;
   			iStateMachine_RWH_CMD := 3050;
   		END_IF;
   
   	3050:
   		// frame a command and send to the DTE.
   		scDTE102_Handling.ActivateCommand.AO	:= 0;
   		scDTE102_Handling.ActivateCommand.WR	:= 0;
   		scDTE102_Handling.ActivateCommand.RD	:= 1;
   		scDTE102_Handling.ActivateCommand.UR	:= 1;
   		scDTE102_Handling.ActivateCommand.ER	:= 1;
   		scDTE102_Handling.ActivateCommand.DR	:= 0;
   		scDTE102_Handling.ActivateCommand.CM	:= 0;
   		INT_TO_BYTE(fb_DataLength);
   		oarsiOutputToDTE[iiOutputStartAdd+2]	:= fb_DataLength.OutUpperNibble;
   		oarsiOutputToDTE[iiOutputStartAdd+3]	:= fb_DataLength.OutLowerNibble;
   		INT_TO_BYTE(fb_DataAddress);
   		oarsiOutputToDTE[iiOutputStartAdd+4]	:= fb_DataAddress.OutUpperNibble;
   		oarsiOutputToDTE[iiOutputStartAdd+5]	:= fb_DataAddress.OutLowerNibble;
   		scDTE102_Handling.ActivateCommand.TR	:= NOT(scDTE102_Handling.Status.TA);
   		odiStatus := 16#7102;
   		iStateMachine_RWH_CMD					:= 3100;
   
   
   	3100:
   
   		IF(scDTE102_Handling.Status.DIAG)THEN		// Error in receiving the data from DTE.
   			oxBusy := 1;
   			oxDone := 0;
   			oxError := 0;
   			scDTE102_Handling.ActivateCommand.AO	:= 0;
   			scDTE102_Handling.ActivateCommand.WR	:= 0;
   			scDTE102_Handling.ActivateCommand.RD	:= 0;
   			scDTE102_Handling.ActivateCommand.UR	:= 0;
   			scDTE102_Handling.ActivateCommand.ER	:= 0;
   			scDTE102_Handling.ActivateCommand.DR	:= 1;
   			scDTE102_Handling.ActivateCommand.CM	:= 0;
   			scDTE102_Handling.ActivateCommand.TR	:= NOT(scDTE102_Handling.Status.TA);
   			odiStatus := 16#7402;
   			iStateMachine_RWH_CMD					:= 19000;
   		ELSE											// ElSE condition, no error then read the status from the DTE.
   			IF(NOT(scDTE102_Handling.Status.TA XOR scDTE102_Handling.ActivateCommand.TR))THEN // Proceed,when TA=TR
   				SINT_TO_INT(fb_SINT_TO_INT,iarsiInputFromDTE[iiInputStartAdd+3]);
   				iRcvdLength := fb_SINT_TO_INT.oINT_var;
   				IF(iRcvdLength = iiRdWrLength)THEN
   					odiStatus := 16#7103;
   					oiRcvdLength := iRcvdLength;
   					CPS(iarsiInputFromDTE[iiInputStartAdd+6],oarsiRcvBuf[0],oiRcvdLength);
   					iStateMachine_RWH_CMD := 13000;
   				ELSIF(NOT(scDTE102_Handling.Status.TP))THEN //Wait until tag comes in field
   					oxBusy := 1;
   					oxDone := 0;
   					oxError := 0;
   					odiStatus := 16#7001;
   					iStateMachine_RWH_CMD := 3100;
   				END_IF;
   			END_IF;
   		END_IF;
   
   
   // Function ID 4 :- read an area of the USER memory of the ID-tag one time
   	4000:
   		// frame a command and send to the DTE.
   		iNoCyclesReqToReadWriteCompleteData := iiRdWrLength/(iSingleCycleDataExchangeLimitInBytes);
   		iLengthToReadWriteInLastCycle := iiRdWrLength MOD (iSingleCycleDataExchangeLimitInBytes);
   		IF iLengthToReadWriteInLastCycle > 0 THEN
   			iNoCyclesReqToReadWriteCompleteData := iNoCyclesReqToReadWriteCompleteData + 1;
   		END_IF;
   
   		iBufferOffset := iiRdWrStartAddr;
   		iRcvdLength := 0;
   		iTotalRcvdLength := 0;
   		odiStatus := 16#7102;
   		iStateMachine_RWH_CMD := 4025;
   
   	4025: //Prepare data to be sent to DTE
   		//Empty the command array for DTE
   		FOR iLoopHandlerVar2 := (iiInputStartAdd + 2) TO (iiInputStartAdd + iSingleCycleDataExchangeLimitInBytes + 6 -1) BY 1 DO;
   	    	oarsiOutputToDTE[iLoopHandlerVar2] := 0;
   	    END_FOR;
   
   		IF(iNoCyclesReqToReadWriteCompleteData > 0)THEN //There are packets, yet to be sent
   
   			fb_DataAddress.Input := iBufferOffset;
   			IF iNoCyclesReqToReadWriteCompleteData <> 1 THEN // Intermediate packet
   				fb_DataLength.Input := iSingleCycleDataExchangeLimitInBytes;
   			ELSE //Last data packet
   				IF iLengthToReadWriteInLastCycle <> 0 THEN
   					fb_DataLength.Input := iLengthToReadWriteInLastCycle;
   				ELSE
   					fb_DataLength.Input := iSingleCycleDataExchangeLimitInBytes;
   				END_IF;
   			END_IF;
   
   			CPS(iarsiSendBuf[iBufferOffset],oarsiOutputToDTE[iiOutputStartAdd+6],fb_DataLength.Input);
   
   			iStateMachine_RWH_CMD := 4050;
   		ELSE (*Operation completed*)
   			IF iTotalRcvdLength = iiRdWrLength THEN
   				iRcvdLength := iTotalRcvdLength;
   				odiStatus := 16#7103;
   				oiRcvdLength := iRcvdLength;
   				iNoCyclesReqToReadWriteCompleteData := 0;
   				iLengthToReadWriteInLastCycle := 0;
   				xMultipleCyclesReq := 0;
   				iBufferOffset := 0;
   				iRcvdLength := 0;
   				iTotalRcvdLength := 0;
   				iStateMachine_RWH_CMD := 18000;
   			ELSE
   				odiStatus := 16#8315; //	Read data: Complete data could not be read
   				iStateMachine_RWH_CMD := 20000;
   			END_IF;
   		END_IF;
   
   
   	4050:
   		// frame a command and send to the DTE.
   		scDTE102_Handling.ActivateCommand.AO	:= 0;
   		scDTE102_Handling.ActivateCommand.WR	:= 0;
   		scDTE102_Handling.ActivateCommand.RD	:= 1;
   		scDTE102_Handling.ActivateCommand.UR	:= 1;
   		scDTE102_Handling.ActivateCommand.ER	:= 0;
   		scDTE102_Handling.ActivateCommand.DR	:= 0;
   		scDTE102_Handling.ActivateCommand.CM	:= 0;
   		INT_TO_BYTE(fb_DataLength);
   		oarsiOutputToDTE[iiOutputStartAdd+2]	:= fb_DataLength.OutUpperNibble;
   		oarsiOutputToDTE[iiOutputStartAdd+3]	:= fb_DataLength.OutLowerNibble;
   		INT_TO_BYTE(fb_DataAddress);
   		oarsiOutputToDTE[iiOutputStartAdd+4]	:= fb_DataAddress.OutUpperNibble;
   		oarsiOutputToDTE[iiOutputStartAdd+5]	:= fb_DataAddress.OutLowerNibble;
   		scDTE102_Handling.ActivateCommand.TR	:= NOT(scDTE102_Handling.Status.TA);
   		odiStatus := 16#7102;
   		iStateMachine_RWH_CMD					:= 4100;
   
   
   	4100:
   		IF(scDTE102_Handling.Status.DIAG)THEN		// Error in receiving the data from DTE.
   		 	oxBusy := 1;
   			oxDone := 0;
   			oxError := 0;
   			scDTE102_Handling.ActivateCommand.AO	:= 0;
   			scDTE102_Handling.ActivateCommand.WR	:= 0;
   			scDTE102_Handling.ActivateCommand.RD	:= 0;
   			scDTE102_Handling.ActivateCommand.UR	:= 0;
   			scDTE102_Handling.ActivateCommand.ER	:= 0;
   			scDTE102_Handling.ActivateCommand.DR	:= 1;
   			scDTE102_Handling.ActivateCommand.CM	:= 0;
   			scDTE102_Handling.ActivateCommand.TR	:= NOT(scDTE102_Handling.Status.TA);
   			odiStatus := 16#7402;
   			iStateMachine_RWH_CMD					:= 19000;
   
   		ELSE											// ElSE condition, no error then read the status from the DTE.
   			IF(NOT(scDTE102_Handling.Status.TA XOR scDTE102_Handling.ActivateCommand.TR))AND(NOT(scDTE102_Handling.Status.CA))THEN
   				//CPSy DTE data to output recieve buffer
   				SINT_TO_INT(fb_SINT_TO_INT,iarsiInputFromDTE[iiInputStartAdd+3]);
   				iRcvdLength := fb_SINT_TO_INT.oINT_var;
   
   					IF iRcvdLength <> fb_DataLength.Input THEN //Device could not write, intended number of data bytes.
   						odiStatus := 16#8315; //	Read data: Complete data could not be read
   						iStateMachine_RWH_CMD := 20000;
   					ELSE //Write successful
   						CPS(iarsiInputFromDTE[iiInputStartAdd+6],oarsiRcvBuf[iTotalRcvdLength],iRcvdLength);
   
   						iTotalRcvdLength := iTotalRcvdLength + iRcvdLength;
   				iBufferOffset := iBufferOffset + iRcvdLength;
   				iNoCyclesReqToReadWriteCompleteData := iNoCyclesReqToReadWriteCompleteData - 1;
   					END_IF;
   				iStateMachine_RWH_CMD := 4025;
   			END_IF;
   		END_IF;
   
   
   
   	// Function ID 5 :- write data to an area of the USER memory of the ID-tag automatically
   	5000:
   		// frame a command and send to the DTE.
   		IF(iiRdWrLength <= (iSingleCycleDataExchangeLimitInBytes))THEN		// Writing in single cycle handling.
   			xMultipleCyclesReq  := 0;
   			fb_DataLength.Input := iiRdWrLength;
   			fb_DataAddress.Input:= iiRdWrStartAddr;
   			CPS(iarsiSendBuf[0],oarsiOutputToDTE[iiOutputStartAdd+6],fb_DataLength.Input);
   			odiStatus := 16#7202;
   			iStateMachine_RWH_CMD := 5050;
   		END_IF;
   
   
   
   	5050:
   		// ElSE condition, no error then frame a command and send to the DTE.
   		scDTE102_Handling.ActivateCommand.AO	:= 0;
   		scDTE102_Handling.ActivateCommand.WR	:= 1;
   		scDTE102_Handling.ActivateCommand.RD	:= 0;
   		scDTE102_Handling.ActivateCommand.UR	:= 1;
   		scDTE102_Handling.ActivateCommand.ER	:= 1;
   		scDTE102_Handling.ActivateCommand.DR	:= 0;
   		scDTE102_Handling.ActivateCommand.CM	:= 0;
   		INT_TO_BYTE(fb_DataLength);
   		oarsiOutputToDTE[iiOutputStartAdd+2]	:= fb_DataLength.OutUpperNibble;
   		oarsiOutputToDTE[iiOutputStartAdd+3]	:= fb_DataLength.OutLowerNibble;
   		INT_TO_BYTE(fb_DataAddress);
   		oarsiOutputToDTE[iiOutputStartAdd+4]	:= fb_DataAddress.OutUpperNibble;
   		oarsiOutputToDTE[iiOutputStartAdd+5]	:= fb_DataAddress.OutLowerNibble;
   		scDTE102_Handling.ActivateCommand.TR	:= NOT(scDTE102_Handling.Status.TA);
   		odiStatus := 16#7202;
   		iStateMachine_RWH_CMD					:= 5100;
   
   
   	5100:
   		IF(scDTE102_Handling.Status.DIAG)THEN		// Error in receiving the data from DTE.
   			oxBusy := 1;
   			oxDone := 0;
   			oxError := 0;
   			scDTE102_Handling.ActivateCommand.AO	:= 0;
   			scDTE102_Handling.ActivateCommand.WR	:= 0;
   			scDTE102_Handling.ActivateCommand.RD	:= 0;
   			scDTE102_Handling.ActivateCommand.UR	:= 0;
   			scDTE102_Handling.ActivateCommand.ER	:= 0;
   			scDTE102_Handling.ActivateCommand.DR	:= 1;
   			scDTE102_Handling.ActivateCommand.CM	:= 0;
   			scDTE102_Handling.ActivateCommand.TR	:= NOT(scDTE102_Handling.Status.TA);
   			odiStatus := 16#7402;
   			iStateMachine_RWH_CMD					:= 19000;
   		ELSE											// ElSE condition, no error then read the status from the DTE.
   			IF(NOT(scDTE102_Handling.Status.TA XOR scDTE102_Handling.ActivateCommand.TR))THEN // Proceed,when TA=TR
   				SINT_TO_INT(fb_SINT_TO_INT,iarsiInputFromDTE[iiInputStartAdd+3]);
   				iRcvdLength := fb_SINT_TO_INT.oINT_var;
   				IF(iRcvdLength = iiRdWrLength)THEN
   					odiStatus := 16#7203;
   					oiRcvdLength := iRcvdLength;
   					iStateMachine_RWH_CMD := 13000;
   				ELSIF(NOT(scDTE102_Handling.Status.TP))THEN
   					oxBusy := 1;
   					oxDone := 0;
   					oxError := 0;
   					odiStatus := 16#7001;
   					iStateMachine_RWH_CMD := 5100;
   				END_IF;
   			END_IF;
   		END_IF;
   
   	// Function ID 6 :- write data to an area of the USER memory of the ID-tag one time
   	6000:
   		// frame a command and send to the DTE.
   		iNoCyclesReqToReadWriteCompleteData := iiRdWrLength/(iSingleCycleDataExchangeLimitInBytes);
   		iLengthToReadWriteInLastCycle := iiRdWrLength MOD (iSingleCycleDataExchangeLimitInBytes);
   		IF iLengthToReadWriteInLastCycle > 0 THEN
   			iNoCyclesReqToReadWriteCompleteData := iNoCyclesReqToReadWriteCompleteData + 1;
   		END_IF;
   
   		iBufferOffset := iiRdWrStartAddr;
   		iRcvdLength := 0;
   		iTotalRcvdLength := 0;
   		odiStatus := 16#7202;
   		iStateMachine_RWH_CMD := 6025;
   
   
   	6025: //Prepare data to be sent to DTE
   		//Empty the command array for DTE
   		FOR iLoopHandlerVar2 := (iiInputStartAdd + 2) TO (iiInputStartAdd + iSingleCycleDataExchangeLimitInBytes + 6 -1) BY 1 DO;
   	    	oarsiOutputToDTE[iLoopHandlerVar2] := 0;
   	    END_FOR;
   
   		IF(iNoCyclesReqToReadWriteCompleteData > 0)THEN //There are packets, yet to be sent
   
   			fb_DataAddress.Input := iBufferOffset;
   			IF iNoCyclesReqToReadWriteCompleteData <> 1 THEN // Intermediate packet
   				fb_DataLength.Input := iSingleCycleDataExchangeLimitInBytes;
   			ELSE //Last data packet
   				IF iLengthToReadWriteInLastCycle <> 0 THEN
   					fb_DataLength.Input := iLengthToReadWriteInLastCycle;
   				ELSE
   					fb_DataLength.Input := iSingleCycleDataExchangeLimitInBytes;
   				END_IF;
   			END_IF;
   
   			CPS(iarsiSendBuf[iTotalRcvdLength],oarsiOutputToDTE[iiOutputStartAdd+6],fb_DataLength.Input);
   
   			iStateMachine_RWH_CMD := 6050;
   		ELSE (*Operation completed*)
   			IF iTotalRcvdLength = iiRdWrLength THEN
   				iRcvdLength := iTotalRcvdLength;
   				odiStatus := 16#7203;
   				oiRcvdLength := iRcvdLength;
   				iNoCyclesReqToReadWriteCompleteData := 0;
   				iLengthToReadWriteInLastCycle := 0;
   				xMultipleCyclesReq := 0;
   				iBufferOffset := 0;
   				iRcvdLength := 0;
   				iTotalRcvdLength := 0;
   
   				iStateMachine_RWH_CMD := 18000;
   			ELSE
   				odiStatus := 16#8316; //	Write data: Complete data could not be written
   				iStateMachine_RWH_CMD := 20000;
   			END_IF;
   		END_IF;
   	6050:
   
   		//Frame a command and send to the DTE.
   		scDTE102_Handling.ActivateCommand.AO	:= 0;
   		scDTE102_Handling.ActivateCommand.WR	:= 1;
   		scDTE102_Handling.ActivateCommand.RD	:= 0;
   		scDTE102_Handling.ActivateCommand.UR	:= 1;
   		scDTE102_Handling.ActivateCommand.ER	:= 0;
   		scDTE102_Handling.ActivateCommand.DR	:= 0;
   		scDTE102_Handling.ActivateCommand.CM	:= 0;
   		INT_TO_BYTE(fb_DataLength);
   		oarsiOutputToDTE[iiOutputStartAdd+2]	:= fb_DataLength.OutUpperNibble;
   		oarsiOutputToDTE[iiOutputStartAdd+3]	:= fb_DataLength.OutLowerNibble;
   		INT_TO_BYTE(fb_DataAddress);
   		oarsiOutputToDTE[iiOutputStartAdd+4]	:= fb_DataAddress.OutUpperNibble;
   		oarsiOutputToDTE[iiOutputStartAdd+5]	:= fb_DataAddress.OutLowerNibble;
   		scDTE102_Handling.ActivateCommand.TR	:= NOT(scDTE102_Handling.Status.TA);
   		odiStatus := 16#7202;
   		iStateMachine_RWH_CMD					:= 6100;
   
   
   	6100:
   		IF(scDTE102_Handling.Status.DIAG)THEN		// Error in receiving the data from DTE.
   			oxBusy := 1;
   			oxDone := 0;
   			oxError := 0;
   			scDTE102_Handling.ActivateCommand.AO	:= 0;
   			scDTE102_Handling.ActivateCommand.WR	:= 0;
   			scDTE102_Handling.ActivateCommand.RD	:= 0;
   			scDTE102_Handling.ActivateCommand.UR	:= 0;
   			scDTE102_Handling.ActivateCommand.ER	:= 0;
   			scDTE102_Handling.ActivateCommand.DR	:= 1;
   			scDTE102_Handling.ActivateCommand.CM	:= 0;
   			scDTE102_Handling.ActivateCommand.TR	:= NOT(scDTE102_Handling.Status.TA);
   			odiStatus := 16#7402;
   			iStateMachine_RWH_CMD					:= 19000;
   
   		ELSE											// ElSE condition, no error then read the status from the DTE.
   			IF(NOT(scDTE102_Handling.Status.TA XOR scDTE102_Handling.ActivateCommand.TR))AND(NOT(scDTE102_Handling.Status.CA))THEN
   				//CPSy DTE data to output recieve buffer
   				SINT_TO_INT(fb_SINT_TO_INT,iarsiInputFromDTE[iiInputStartAdd+3]);
   				iRcvdLength := fb_SINT_TO_INT.oINT_var;
   
   					IF iRcvdLength <> fb_DataLength.Input THEN //Device could not write, intended number of data bytes.
   						odiStatus := 16#8316; //	Write data: Complete data could not be written
   						iStateMachine_RWH_CMD := 20000;
   					ELSE //Write successful
   						CPS(iarsiInputFromDTE[iiInputStartAdd+6],oarsiRcvBuf[iTotalRcvdLength],iRcvdLength);
   
   						iTotalRcvdLength := iTotalRcvdLength + iRcvdLength;
   						iBufferOffset := iBufferOffset + iRcvdLength;
   						iNoCyclesReqToReadWriteCompleteData := iNoCyclesReqToReadWriteCompleteData - 1;
   					END_IF;
   				iStateMachine_RWH_CMD := 6025;
   			END_IF;
   		END_IF;
   
   
   
   	// Function ID 7 :- write data verified to an area of the USER memory of the ID-tag automatically
   	7000:
   		// frame a command and send to the DTE.
   		IF(iiRdWrLength <= (iSingleCycleDataExchangeLimitInBytes))THEN		// Writing in single cycle handling.
   			xMultipleCyclesReq  := 0;
   			fb_DataLength.Input := iiRdWrLength;
   			fb_DataAddress.Input:= iiRdWrStartAddr;
   			CPS(iarsiSendBuf[0],oarsiOutputToDTE[iiOutputStartAdd+6],fb_DataLength.Input);
   			odiStatus := 16#7202;
   			iStateMachine_RWH_CMD := 7050;
   		END_IF;
   
   
   
   	7050:
   		// ElSE condition, no error then frame a command and send to the DTE.
   		scDTE102_Handling.ActivateCommand.AO	:= 0;
   		scDTE102_Handling.ActivateCommand.WR	:= 1;
   		scDTE102_Handling.ActivateCommand.RD	:= 1;
   		scDTE102_Handling.ActivateCommand.UR	:= 1;
   		scDTE102_Handling.ActivateCommand.ER	:= 1;
   		scDTE102_Handling.ActivateCommand.DR	:= 0;
   		scDTE102_Handling.ActivateCommand.CM	:= 0;
   		INT_TO_BYTE(fb_DataLength);
   		oarsiOutputToDTE[iiOutputStartAdd+2]	:= fb_DataLength.OutUpperNibble;
   		oarsiOutputToDTE[iiOutputStartAdd+3]	:= fb_DataLength.OutLowerNibble;
   		INT_TO_BYTE(fb_DataAddress);
   		oarsiOutputToDTE[iiOutputStartAdd+4]	:= fb_DataAddress.OutUpperNibble;
   		oarsiOutputToDTE[iiOutputStartAdd+5]	:= fb_DataAddress.OutLowerNibble;
   		scDTE102_Handling.ActivateCommand.TR	:= NOT(scDTE102_Handling.Status.TA);
   		odiStatus := 16#7202;
   		iStateMachine_RWH_CMD					:= 7100;
   
   
   	7100:
   		IF(scDTE102_Handling.Status.DIAG)THEN		// Error in receiving the data from DTE.
   			oxBusy := 1;
   			oxDone := 0;
   			oxError := 0;
   			scDTE102_Handling.ActivateCommand.AO	:= 0;
   			scDTE102_Handling.ActivateCommand.WR	:= 0;
   			scDTE102_Handling.ActivateCommand.RD	:= 0;
   			scDTE102_Handling.ActivateCommand.UR	:= 0;
   			scDTE102_Handling.ActivateCommand.ER	:= 0;
   			scDTE102_Handling.ActivateCommand.DR	:= 1;
   			scDTE102_Handling.ActivateCommand.CM	:= 0;
   			scDTE102_Handling.ActivateCommand.TR	:= NOT(scDTE102_Handling.Status.TA);
   			odiStatus := 16#7402;
   			iStateMachine_RWH_CMD					:= 19000;
   		ELSE											// ElSE condition, no error then read the status from the DTE.
   			IF(NOT(scDTE102_Handling.Status.TA XOR scDTE102_Handling.ActivateCommand.TR))AND(NOT(scDTE102_Handling.Status.CA))THEN
   				SINT_TO_INT(fb_SINT_TO_INT,iarsiInputFromDTE[iiInputStartAdd+3]);
   				iRcvdLength := fb_SINT_TO_INT.oINT_var;
   				IF(iRcvdLength = iiRdWrLength)THEN
   					odiStatus := 16#7203;
   					oiRcvdLength := iRcvdLength;
   					CPS(iarsiInputFromDTE[iiInputStartAdd+6],oarsiRcvBuf[0],oiRcvdLength);
   					iStateMachine_RWH_CMD := 13000;
   				ELSIF(NOT(scDTE102_Handling.Status.TP))THEN
   					oxBusy := 1;
   					oxDone := 0;
   					oxError := 0;
   					odiStatus := 16#7001;
   					iStateMachine_RWH_CMD := 7100;
   				END_IF;
   			END_IF;
   		END_IF;
   
   	// Function ID 8 :- write data verified to an area of the USER memory of the ID-tag one time
   	8000:
   		// frame a command and send to the DTE.
   		iNoCyclesReqToReadWriteCompleteData := iiRdWrLength/(iSingleCycleDataExchangeLimitInBytes);
   		iLengthToReadWriteInLastCycle := iiRdWrLength MOD (iSingleCycleDataExchangeLimitInBytes);
   		IF iLengthToReadWriteInLastCycle > 0 THEN
   			iNoCyclesReqToReadWriteCompleteData := iNoCyclesReqToReadWriteCompleteData + 1;
   		END_IF;
   
   		iBufferOffset := iiRdWrStartAddr;
   		iRcvdLength := 0;
   		iTotalRcvdLength := 0;
   		odiStatus := 16#7202;
   		iStateMachine_RWH_CMD := 8025;
   
   
   	8025: //Prepare data to be sent to DTE
   		//Empty the command array for DTE
   		FOR iLoopHandlerVar2 := (iiInputStartAdd + 2) TO (iiInputStartAdd + iSingleCycleDataExchangeLimitInBytes + 6 -1) BY 1 DO;
   	    	oarsiOutputToDTE[iLoopHandlerVar2] := 0;
   	    END_FOR;
   
   		IF(iNoCyclesReqToReadWriteCompleteData > 0)THEN //There are packets, yet to be sent
   
   			fb_DataAddress.Input := iBufferOffset;
   			IF iNoCyclesReqToReadWriteCompleteData <> 1 THEN // Intermediate packet
   				fb_DataLength.Input := iSingleCycleDataExchangeLimitInBytes;
   			ELSE //Last data packet
   				IF iLengthToReadWriteInLastCycle <> 0 THEN
   					fb_DataLength.Input := iLengthToReadWriteInLastCycle;
   				ELSE
   					fb_DataLength.Input := iSingleCycleDataExchangeLimitInBytes;
   				END_IF;
   			END_IF;
   
   			CPS(iarsiSendBuf[iTotalRcvdLength],oarsiOutputToDTE[iiOutputStartAdd+6],fb_DataLength.Input);
   
   			iStateMachine_RWH_CMD := 8050;
   
   
   		ELSE (*Operation completed*)
   			IF iTotalRcvdLength = iiRdWrLength THEN
   				iRcvdLength := iTotalRcvdLength;
   				odiStatus := 16#7203;
   				oiRcvdLength := iRcvdLength;
   				iNoCyclesReqToReadWriteCompleteData := 0;
   				iLengthToReadWriteInLastCycle := 0;
   				xMultipleCyclesReq := 0;
   				iBufferOffset := 0;
   				iRcvdLength := 0;
   				iTotalRcvdLength := 0;
   				iStateMachine_RWH_CMD := 18000;
   			ELSE
   				odiStatus := 16#8313; //	Write-verified: Complete data could not be written
   				iStateMachine_RWH_CMD := 20000;
   			END_IF;
   		END_IF;
   
   
   	8050:
   		//Frame a command and send to the DTE.
   		scDTE102_Handling.ActivateCommand.AO	:= 0;
   		scDTE102_Handling.ActivateCommand.WR	:= 1;
   		scDTE102_Handling.ActivateCommand.RD	:= 1;
   		scDTE102_Handling.ActivateCommand.UR	:= 1;
   		scDTE102_Handling.ActivateCommand.ER	:= 0;
   		scDTE102_Handling.ActivateCommand.DR	:= 0;
   		scDTE102_Handling.ActivateCommand.CM	:= 0;
   		INT_TO_BYTE(fb_DataLength);
   		oarsiOutputToDTE[iiOutputStartAdd+2]	:= fb_DataLength.OutUpperNibble;
   		oarsiOutputToDTE[iiOutputStartAdd+3]	:= fb_DataLength.OutLowerNibble;
   		INT_TO_BYTE(fb_DataAddress);
   		oarsiOutputToDTE[iiOutputStartAdd+4]	:= fb_DataAddress.OutUpperNibble;
   		oarsiOutputToDTE[iiOutputStartAdd+5]	:= fb_DataAddress.OutLowerNibble;
   		scDTE102_Handling.ActivateCommand.TR	:= NOT(scDTE102_Handling.Status.TA);
   		odiStatus := 16#7202;
   		iStateMachine_RWH_CMD					:= 8100;
   
   
   	8100:
   		IF(scDTE102_Handling.Status.DIAG)THEN		// Error in receiving the data from DTE.
   			oxBusy := 1;
   			oxDone := 0;
   			oxError := 0;
   			scDTE102_Handling.ActivateCommand.AO	:= 0;
   			scDTE102_Handling.ActivateCommand.WR	:= 0;
   			scDTE102_Handling.ActivateCommand.RD	:= 0;
   			scDTE102_Handling.ActivateCommand.UR	:= 0;
   			scDTE102_Handling.ActivateCommand.ER	:= 0;
   			scDTE102_Handling.ActivateCommand.DR	:= 1;
   			scDTE102_Handling.ActivateCommand.CM	:= 0;
   			scDTE102_Handling.ActivateCommand.TR	:= NOT(scDTE102_Handling.Status.TA);
   			odiStatus := 16#7402;
   			iStateMachine_RWH_CMD					:= 19000;
   		ELSE											// ElSE condition, no error then read the status from the DTE.
   			IF(NOT(scDTE102_Handling.Status.TA XOR scDTE102_Handling.ActivateCommand.TR))AND(NOT(scDTE102_Handling.Status.CA))THEN
   				//CPSy DTE data to output recieve buffer
   				SINT_TO_INT(fb_SINT_TO_INT,iarsiInputFromDTE[iiInputStartAdd+3]);
   				iRcvdLength := fb_SINT_TO_INT.oINT_var;
   
   					IF iRcvdLength <> fb_DataLength.Input THEN //Device could not write, intended number of data bytes.
   						odiStatus := 16#8313; 	//Write-verified: Complete data could not be written
   						iStateMachine_RWH_CMD := 20000;
   					ELSE //Write successful
   					CPS(iarsiInputFromDTE[iiInputStartAdd+6],oarsiRcvBuf[iTotalRcvdLength],iRcvdLength);
   
   						iTotalRcvdLength := iTotalRcvdLength + iRcvdLength;
   						iBufferOffset := iBufferOffset + iRcvdLength;
   						iNoCyclesReqToReadWriteCompleteData := iNoCyclesReqToReadWriteCompleteData - 1;
   					END_IF;
   				iStateMachine_RWH_CMD := 8025;
   			END_IF;
   		END_IF;
   
   	// Function ID 9 :- switch off the antenna field of the RFID-Read/Write Head
   	9000:
   		// ElSE condition, no error then frame a command and send to the DTE.
   		scDTE102_Handling.ActivateCommand.AO	:= 1;
   		scDTE102_Handling.ActivateCommand.WR	:= 0;
   		scDTE102_Handling.ActivateCommand.RD	:= 0;
   		scDTE102_Handling.ActivateCommand.UR	:= 0;
   		scDTE102_Handling.ActivateCommand.ER	:= 0;
   		scDTE102_Handling.ActivateCommand.DR	:= 0;
   		scDTE102_Handling.ActivateCommand.CM	:= 0;
   		scDTE102_Handling.ActivateCommand.TR	:= NOT(scDTE102_Handling.Status.TA);
   		odiStatus := 16#7501;
   		iStateMachine_RWH_CMD					:= 9050;
   
   
   	9050:
   		IF(scDTE102_Handling.Status.DIAG)THEN		// Error in receiving the data from DTE.
   			oxBusy := 1;
   			oxDone := 0;
   			oxError := 0;
   			scDTE102_Handling.ActivateCommand.AO	:= 0;
   			scDTE102_Handling.ActivateCommand.WR	:= 0;
   			scDTE102_Handling.ActivateCommand.RD	:= 0;
   			scDTE102_Handling.ActivateCommand.UR	:= 0;
   			scDTE102_Handling.ActivateCommand.ER	:= 0;
   			scDTE102_Handling.ActivateCommand.DR	:= 1;
   			scDTE102_Handling.ActivateCommand.CM	:= 0;
   			scDTE102_Handling.ActivateCommand.TR	:= NOT(scDTE102_Handling.Status.TA);
   			odiStatus := 16#7402;
   			iStateMachine_RWH_CMD					:= 19000;
   		ELSE											// ElSE condition, no error then read the status from the DTE.
   			IF(NOT(scDTE102_Handling.Status.TA XOR scDTE102_Handling.ActivateCommand.TR))AND(scDTE102_Handling.Status.AI)THEN
   				oxBusy := 0;
   				oxDone := 1;
   				oxError := 0;
   				odiStatus := 16#7502;
   				iStateMachine_RWH_CMD				:= 25000;
   			END_IF;
   		END_IF;
   
   
   	// Function ID 10 :- Switch Antenna ON Command
   	10000:
   		//no error then frame a command and send to the DTE.
   		// Antenna will be switched ON
   		scDTE102_Handling.ActivateCommand.AO	:= 0;
   		scDTE102_Handling.ActivateCommand.WR	:= 0;
   		scDTE102_Handling.ActivateCommand.RD	:= 0;
   		scDTE102_Handling.ActivateCommand.UR	:= 0;
   		scDTE102_Handling.ActivateCommand.ER	:= 0;
   		scDTE102_Handling.ActivateCommand.DR	:= 0;
   		scDTE102_Handling.ActivateCommand.CM	:= 0;
   		scDTE102_Handling.ActivateCommand.TR	:= NOT(scDTE102_Handling.Status.TA);
   		odiStatus := 16#7601;
   		iStateMachine_RWH_CMD					:= 10050;
   
   
   	10050:
   		IF(scDTE102_Handling.Status.DIAG)THEN		// Error in receiving the data from DTE.
   			oxBusy := 1;
   			oxDone := 0;
   			oxError := 0;
   			scDTE102_Handling.ActivateCommand.AO	:= 0;
   			scDTE102_Handling.ActivateCommand.WR	:= 0;
   			scDTE102_Handling.ActivateCommand.RD	:= 0;
   			scDTE102_Handling.ActivateCommand.UR	:= 0;
   			scDTE102_Handling.ActivateCommand.ER	:= 0;
   			scDTE102_Handling.ActivateCommand.DR	:= 1;
   			scDTE102_Handling.ActivateCommand.CM	:= 0;
   			scDTE102_Handling.ActivateCommand.TR	:= NOT(scDTE102_Handling.Status.TA);
   			odiStatus := 16#7402;
   			iStateMachine_RWH_CMD					:= 19000;
   		ELSE											// ElSE condition, no error then read the status from the DTE.
   			IF(NOT(scDTE102_Handling.Status.TA XOR scDTE102_Handling.ActivateCommand.TR))AND(NOT(scDTE102_Handling.Status.AI))THEN
   				odiStatus := 16#7602;
   				iStateMachine_RWH_CMD				:= 18000;
   			END_IF;
   		END_IF;
   
   
   
   
   	// Function ID 11 :- execute a command to read device parameters one time
   	11000:
   		// frame a command and send to the DTE.
   		scDTE102_Handling.ActivateCommand.AO	:= 0;
   		scDTE102_Handling.ActivateCommand.WR	:= 0;
   		scDTE102_Handling.ActivateCommand.RD	:= 1;
   		scDTE102_Handling.ActivateCommand.UR	:= 0;
   		scDTE102_Handling.ActivateCommand.ER	:= 0;
   		scDTE102_Handling.ActivateCommand.DR	:= 0;
   		scDTE102_Handling.ActivateCommand.CM	:= 1;
   		IF(iCmdCode >= 16#62C8 AND iCmdCode <= 16#62D0)THEN
   			oarsiOutputToDTE[iiOutputStartAdd+2]					:= 0;
   			oarsiOutputToDTE[iiOutputStartAdd+3]					:= 16#02;
   		ELSE
   			oarsiOutputToDTE[iiOutputStartAdd+2]					:= 0;
   			oarsiOutputToDTE[iiOutputStartAdd+3]					:= 16#06;
   		END_IF;
   		fb_CmdCode.Input := iCmdCode;
   		INT_TO_BYTE(fb_CmdCode);
   		oarsiOutputToDTE[iiOutputStartAdd+4]						:= fb_CmdCode.OutUpperNibble;
   		oarsiOutputToDTE[iiOutputStartAdd+5]						:= fb_CmdCode.OutLowerNibble;
   
   		IF(iCmdCode = 16#62D1)THEN
   			fb_DataAddress.Input									:= iiRdWrStartAddr;
   			INT_TO_BYTE(fb_DataAddress);
   			oarsiOutputToDTE[iiOutputStartAdd+6]					:= fb_DataAddress.OutUpperNibble;
   			oarsiOutputToDTE[iiOutputStartAdd+7]					:= fb_DataAddress.OutLowerNibble;
   			fb_DataLength.Input										:= iiRdWrLength;
   			INT_TO_BYTE(fb_DataLength);
   			oarsiOutputToDTE[iiOutputStartAdd+8]					:= fb_DataLength.OutUpperNibble;
   			oarsiOutputToDTE[iiOutputStartAdd+9]					:= fb_DataLength.OutLowerNibble;
   		ELSE
   			oarsiOutputToDTE[iiOutputStartAdd+6]					:= 0;
   			oarsiOutputToDTE[iiOutputStartAdd+7]					:= 0;
   			oarsiOutputToDTE[iiOutputStartAdd+8]					:= 0;
   			oarsiOutputToDTE[iiOutputStartAdd+9]					:= 0;
   		END_IF;
   
   		scDTE102_Handling.ActivateCommand.TR	:= NOT(scDTE102_Handling.Status.TA);
   		odiStatus := 16#7701;
   		iStateMachine_RWH_CMD					:= 11050;
   
   	11050:
   		IF(scDTE102_Handling.Status.DIAG)AND(iCmdCode<>16#62C8)THEN		// Error in receiving  the data from DTE.
   			oxBusy := 1;
   			oxDone := 0;
   			oxError := 0;
   			scDTE102_Handling.ActivateCommand.AO	:= 0;
   			scDTE102_Handling.ActivateCommand.WR	:= 0;
   			scDTE102_Handling.ActivateCommand.RD	:= 1;
   			scDTE102_Handling.ActivateCommand.UR	:= 0;
   			scDTE102_Handling.ActivateCommand.ER	:= 0;
   			scDTE102_Handling.ActivateCommand.DR	:= 0;
   			scDTE102_Handling.ActivateCommand.CM	:= 1;
   			oarsiOutputToDTE[iiOutputStartAdd+2]	:= 0;
   			oarsiOutputToDTE[iiOutputStartAdd+3]	:= 16#02;
   			oarsiOutputToDTE[iiOutputStartAdd+4]	:= 16#62;
   			oarsiOutputToDTE[iiOutputStartAdd+5]	:= 16#C8;
   			scDTE102_Handling.ActivateCommand.TR	:= NOT(scDTE102_Handling.Status.TA);
   			odiStatus := 16#7402;
   			iStateMachine_RWH_CMD					:= 19000;
   		ELSE										// ElSE condition, no error then read the status from the DTE.
   			IF(NOT(scDTE102_Handling.Status.TA XOR scDTE102_Handling.ActivateCommand.TR))AND(scDTE102_Handling.Status.CA)THEN
   				IF(iCmdCode = 16#62C8)THEN
   					SINT_TO_INT(fb_SINT_TO_INT,iarsiInputFromDTE[iiInputStartAdd+7]);
   					oiRcvdLength := fb_SINT_TO_INT.oINT_var;
   
   					iRcvdLength := fb_SINT_TO_INT.oINT_var * 4;
   					CPS(iarsiInputFromDTE[iiInputStartAdd+8],oarsiRcvBuf[0],iRcvdLength);
   				ELSIF(iCmdCode = 16#62C9)THEN
   					oiRcvdLength := 6;
   					oarsiRcvBuf[0] := iarsiInputFromDTE[iiInputStartAdd+6];
   					oarsiRcvBuf[1] := iarsiInputFromDTE[iiInputStartAdd+7];
   					oarsiRcvBuf[2] := iarsiInputFromDTE[iiInputStartAdd+8];
   					oarsiRcvBuf[3] := iarsiInputFromDTE[iiInputStartAdd+9];
   					oarsiRcvBuf[4] := iarsiInputFromDTE[iiInputStartAdd+10];
   					oarsiRcvBuf[5] := iarsiInputFromDTE[iiInputStartAdd+11];
   				ELSIF(iCmdCode = 16#62CD)THEN
   					SINT_TO_INT(fb_SINT_TO_INT,iarsiInputFromDTE[iiInputStartAdd+7]);
   					iRcvdLength := fb_SINT_TO_INT.oINT_var;
   
   					oiRcvdLength := iRcvdLength;
   					CPS(iarsiInputFromDTE[iiInputStartAdd+8],oarsiRcvBuf[0],iRcvdLength);
   				ELSIF(iCmdCode = 16#62CE)THEN
   					SINT_TO_INT(fb_SINT_TO_INT,iarsiInputFromDTE[iiInputStartAdd+7]);
   					iRcvdLength := fb_SINT_TO_INT.oINT_var;
   
   					oiRcvdLength := iRcvdLength;
   					oarsiRcvBuf[0] := iarsiInputFromDTE[iiInputStartAdd+8];
   					oarsiRcvBuf[1] := iarsiInputFromDTE[iiInputStartAdd+9];
   					oarsiRcvBuf[2] := iarsiInputFromDTE[iiInputStartAdd+10];
   					oarsiRcvBuf[3] := iarsiInputFromDTE[iiInputStartAdd+11];
   					oarsiRcvBuf[4] := iarsiInputFromDTE[iiInputStartAdd+12];
   				ELSIF(iCmdCode = 16#62CF)THEN
   					oiRcvdLength := 1;
   					oarsiRcvBuf[0] := iarsiInputFromDTE[iiInputStartAdd+7];
   				ELSIF(iCmdCode = 16#62D0)THEN
   					oiRcvdLength := 1;
   					oarsiRcvBuf[0] := iarsiInputFromDTE[iiInputStartAdd+7];
   				ELSIF(iCmdCode = 16#62D1)THEN
   					SINT_TO_INT(fb_SINT_TO_INT,iarsiInputFromDTE[iiInputStartAdd+7]);
   					iRcvdLength := fb_SINT_TO_INT.oINT_var;
   
   					oiRcvdLength := iRcvdLength;
   					CPS(iarsiInputFromDTE[iiInputStartAdd+8],oarsiRcvBuf[0],oiRcvdLength);
   				ELSIF(iCmdCode = 16#62D2)THEN
   					oiRcvdLength := 1;
   					oarsiRcvBuf[0] := iarsiInputFromDTE[iiInputStartAdd+7];
   				ELSIF(iCmdCode = 16#62D3)THEN
   					oiRcvdLength := 1;
   					oarsiRcvBuf[0] := iarsiInputFromDTE[iiInputStartAdd+7];
   				END_IF;
   				odiStatus := 16#7702;
   				iStateMachine_RWH_CMD := 18000;
   			END_IF;
   		END_IF;
   
   
   	// Function ID 12 :- execute a command to set device parameters one time
   	12000:
   		// frame a command and send to the DTE.
   		scDTE102_Handling.ActivateCommand.AO	:= 0;
   		scDTE102_Handling.ActivateCommand.WR	:= 1;
   		scDTE102_Handling.ActivateCommand.RD	:= 0;
   		scDTE102_Handling.ActivateCommand.UR	:= 0;
   		scDTE102_Handling.ActivateCommand.ER	:= 0;
   		scDTE102_Handling.ActivateCommand.DR	:= 0;
   		scDTE102_Handling.ActivateCommand.CM	:= 1;
   		IF(iCmdCode = 16#65D8)THEN
   			oarsiOutputToDTE[iiOutputStartAdd+2]					:= 0;
   			oarsiOutputToDTE[iiOutputStartAdd+3]					:= 16#06;
   		ELSIF(iCmdCode = 16#65DC OR iCmdCode = 16#65DD)THEN
   			oarsiOutputToDTE[iiOutputStartAdd+2]					:= 0;
   			oarsiOutputToDTE[iiOutputStartAdd+3]					:= 16#02;
   		ELSE
   			oarsiOutputToDTE[iiOutputStartAdd+2]					:= 0;
   			oarsiOutputToDTE[iiOutputStartAdd+3]					:= 16#04;
   		END_IF;
   		fb_CmdCode.Input := iCmdCode;
   		INT_TO_BYTE(fb_CmdCode);
   		oarsiOutputToDTE[iiOutputStartAdd+4]						:= fb_CmdCode.OutUpperNibble;
   		oarsiOutputToDTE[iiOutputStartAdd+5]						:= fb_CmdCode.OutLowerNibble;
   
   		IF(iCmdCode = 16#65D8)THEN
   			fb_DataAddress.Input									:= iiRdWrStartAddr;
   			INT_TO_BYTE(fb_DataAddress);
   			oarsiOutputToDTE[iiOutputStartAdd+6]					:= fb_DataAddress.OutUpperNibble;
   			oarsiOutputToDTE[iiOutputStartAdd+7]					:= fb_DataAddress.OutLowerNibble;
   			fb_DataLength.Input										:= iiRdWrLength;
   			INT_TO_BYTE(fb_DataLength);
   			oarsiOutputToDTE[iiOutputStartAdd+8]					:= fb_DataLength.OutUpperNibble;
   			oarsiOutputToDTE[iiOutputStartAdd+9]					:= fb_DataLength.OutLowerNibble;
   		ELSE
   			oarsiOutputToDTE[iiOutputStartAdd+6]					:= 0;
   			oarsiOutputToDTE[iiOutputStartAdd+7]					:= iarsiSendBuf[0];
   			oarsiOutputToDTE[iiOutputStartAdd+8]					:= 0;
   			oarsiOutputToDTE[iiOutputStartAdd+9]					:= 0;
   		END_IF;
   
   		scDTE102_Handling.ActivateCommand.TR	:= NOT(scDTE102_Handling.Status.TA);
   		odiStatus := 16#7801;
   		iStateMachine_RWH_CMD					:= 12050;
   
   	12050:
   		IF(scDTE102_Handling.Status.DIAG)THEN		// Error in receiving  the data from DTE.
   			oxBusy := 1;
   			oxDone := 0;
   			oxError := 0;
   			scDTE102_Handling.ActivateCommand.AO	:= 0;
   			scDTE102_Handling.ActivateCommand.WR	:= 0;
   			scDTE102_Handling.ActivateCommand.RD	:= 1;
   			scDTE102_Handling.ActivateCommand.UR	:= 0;
   			scDTE102_Handling.ActivateCommand.ER	:= 0;
   			scDTE102_Handling.ActivateCommand.DR	:= 0;
   			scDTE102_Handling.ActivateCommand.CM	:= 1;
   			oarsiOutputToDTE[iiOutputStartAdd+2]	:= 0;
   			oarsiOutputToDTE[iiOutputStartAdd+3]	:= 16#02;
   			oarsiOutputToDTE[iiOutputStartAdd+4]	:= 16#62;
   			oarsiOutputToDTE[iiOutputStartAdd+5]	:= 16#C8;
   			scDTE102_Handling.ActivateCommand.TR	:= NOT(scDTE102_Handling.Status.TA);
   			odiStatus := 16#7402;
   			iStateMachine_RWH_CMD					:= 19000;
   		ELSE										// ElSE condition, no error then read the status from the DTE.
   			IF(NOT(scDTE102_Handling.Status.TA XOR scDTE102_Handling.ActivateCommand.TR))AND(scDTE102_Handling.Status.CA)THEN
   				IF(iCmdCode >= 16#65D6 AND iCmdCode <= 16#65DB)THEN
   					oiRcvdLength := 1;
   					oarsiRcvBuf[0] := iarsiInputFromDTE[iiInputStartAdd+7];
   				ELSIF(iCmdCode = 16#65DC OR iCmdCode = 16#65DD)THEN
   					oiRcvdLength := 0;
   					FOR iLoopHandlerVar1 := 0 TO (iActSizeOfRcvBuf-1) BY 1 DO;
   						oarsiRcvBuf[iLoopHandlerVar1] := 0;
   						iLoopHandlerVar1 := 0;
   					END_FOR;
   				END_IF;
   
   				odiStatus := 16#7802;
   				iStateMachine_RWH_CMD := 18000;
   			END_IF;
   		END_IF;
   
   
   	// Keep alive asynchronous command if only parameters are changed or same or other tag comes again in front of antenna
   	13000:
   
   		IF(fb_OSRI_TagPresent.OutputBit)AND(ixExecute)AND(NOT(oxError))THEN
               IF(iActSizeOfInputFromDTE <> iActSizeOfOutputToDTE)THEN
                   odiStatus := 16#8104; //Different sizes of the iarsiInputFromDTE input parameter and oarsiOutputToDTE output parameter                                                                    // Input and output data sizes not equal.
                   iStateMachine_RWH_CMD := 20000;
   			ELSIF(isiModuleID < 12 OR isiModuleID > 19)THEN
   				odiStatus := 16#8112;					// Wrong Module ID entered by user.
   				iStateMachine_RWH_CMD := 20000;
   			ELSIF(iiInputStartAdd < iLowerLimitInputStartAdd OR iiInputStartAdd > iUpperLimitInputStopAdderess)THEN
   				odiStatus := 16#8113;					// Wrong Input Start Address entered by user.
   				iStateMachine_RWH_CMD := 20000;
   			ELSIF(iiOutputStartAdd < iLowerLimitOutputStartAdd OR iiOutputStartAdd > iUpperLimitOutputStopAdderess)THEN
   				odiStatus := 16#8114;					// Wrong Output Start Address entered by user.
   				iStateMachine_RWH_CMD := 20000;
               ELSIF((iiRdWrLength < 1 or iiRdWrLength > iActSizeOfRcvBuf)AND(isiFunctionID <> 9 AND isiFunctionID <> 10 AND isiFunctionID <> 1 AND isiFunctionID <> 2 AND isiFunctionID <> 11 AND isiFunctionID <> 12)) OR
                   ((iiRdWrLength < 1 or iiRdWrLength > iActSizeOfRcvBuf) AND((isiFunctionID = 11 AND iiCmdCode = 16#62D1)OR(isiFunctionID = 12 AND iiCmdCode = 16#65D8)))THEN
                   odiStatus := 16#8305;                        // iiRdWrLength input parameter <= 0 or greater than the defined receive buffer (oarsiRcvBuf)
                   iStateMachine_RWH_CMD := 20000;
               ELSIF((iiRdWrLength < 1 or iiRdWrLength > iActSizeOfSendBuf)AND(isiFunctionID <> 9 AND isiFunctionID <> 10 AND isiFunctionID <> 1 AND isiFunctionID <> 2 AND isiFunctionID <> 11 AND isiFunctionID <> 12)) OR
                   ((iiRdWrLength < 1 or iiRdWrLength > iActSizeOfSendBuf) AND((isiFunctionID = 11 AND iiCmdCode = 16#62D1)OR(isiFunctionID = 12 AND iiCmdCode = 16#65D8)))THEN
                   odiStatus := 16#8306; 						// iiRdWrLength input parameter <= 0 or greater than the defined send buffer (iarsiSendBuf)
                   iStateMachine_RWH_CMD := 20000;
               ELSIF(iiRdWrLength < 1 or iiRdWrLength > (iSingleCycleDataExchangeLimitInBytes))AND((isiFunctionID = 3)OR(isiFunctionID = 5)OR(isiFunctionID = 7))THEN
                   odiStatus := 16#8307;                                                                     // Invalid Read Write data length if asynchronous command is selected.
                   iStateMachine_RWH_CMD := 20000;
               ELSIF((iiRdWrStartAddr < 0 OR iiRdWrStartAddr > (iActSizeOfSendBuf-iiRdWrLength))AND(isiFunctionID <> 9 AND isiFunctionID <> 10 AND isiFunctionID <> 1 AND isiFunctionID <> 2 AND isiFunctionID <> 11 AND isiFunctionID <> 12)) OR
                    ((iiRdWrStartAddr < 0 OR iiRdWrStartAddr > (iActSizeOfSendBuf-iiRdWrLength)) AND((isiFunctionID = 11 AND iiCmdCode = 16#62D1)OR(isiFunctionID = 12 AND iiCmdCode = 16#65D8)))THEN
                   odiStatus := 16#8109;                                                                     // iiRdWrStartAddr input is invalid
                   iStateMachine_RWH_CMD := 20000;
               ELSE
                   oxBusy := 1;
                   oxDone := 0;
                   oxError := 0;
                   odiStatus := 16#0000;
                   iStateMachine_RWH_CMD := siActiveFunctionID * ciStateMachineSeparator;
               END_IF;
   		ELSIF(NOT(oxTagPresent))AND(ixExecute)THEN
   	            oxBusy := 1;
   	            oxDone := 0;
   	            oxError := 0;
   	            odiStatus := 16#7001;
   	            oiRcvdLength := 0;
   	            oiDiagLength := 0;
   	            ardiDiagData[0] := 0;
   	            ardiDiagData[1] := 0;
   	            ardiDiagData[2] := 0;
   	            ardiDiagData[3] := 0;
   	            oardiDiagData[0] := 0;
   	            oardiDiagData[1] := 0;
   	            oardiDiagData[2] := 0;
   	            oardiDiagData[3] := 0;
   	            fb_DataLength.Input := 0;
   	            INT_TO_BYTE(fb_DataLength);
   	            fb_DataAddress.Input := 0;
   	            INT_TO_BYTE(fb_DataAddress);
   
   				FOR iLoopHandlerVar1 :=0 TO (iActSizeOfRcvBuf-1) BY 1 DO;
   	               oarsiRcvBuf[iLoopHandlerVar1] := 0;
   	            END_FOR;
   	            FOR iLoopHandlerVar2 := (iiInputStartAdd + 2) TO (iiInputStartAdd + iSingleCycleDataExchangeLimitInBytes + 6 -1) BY 1 DO;
   	               oarsiOutputToDTE[iLoopHandlerVar2] := 0;
   	            END_FOR;
   
   	            iLoopHandlerVar1 := 0;
   	            iLoopHandlerVar2 := 0;
   	            iNoCyclesReqToReadWriteCompleteData := 0;
   	            iLengthToReadWriteInLastCycle := 0;
   	            xMultipleCyclesReq := 0;
   	            iBufferOffset := 0;
   	            iRcvdLength := 0;
   				iTotalRcvdLength := 0;
   				fb_SINT_TO_INT.iSINT_var := 0;
   				SINT_TO_INT(fb_SINT_TO_INT,fb_SINT_TO_INT.iSINT_var);
   	            iStateMachine_RWH_CMD := 13000;
   		ELSIF(NOT(ixExecute))THEN
   	            oxBusy := 0;
   	            oxDone := 0;
   	            oxError := 0;
   	            odiStatus := 16#0000;
   	            iStateMachine_RWH_CMD := 25000;
   		ELSIF(ixExecute)THEN
   	            oxBusy := 0;
   	            oxDone := 1;
   	            oxError := 0;
   	            odiStatus := 16#0000;
   	            iStateMachine_RWH_CMD := 13000;
   		END_IF;
   
   
   	//Report successful operation
   	18000:
   		oxBusy := 0;
   		oxDone := 1;
   		oxError := 0;
   		odiStatus := 16#0000;
   		iStateMachine_RWH_CMD := 25000;
   
   
   	// Diagnostics read Step
   	19000:
   		IF(NOT(scDTE102_Handling.Status.TA XOR scDTE102_Handling.ActivateCommand.TR))THEN // Proceed,when TA=TR
   			odiStatus := 16#7403;
   			IF(siActiveFunctionID = 11 OR siActiveFunctionID = 12)THEN
   				oiDiagLength := oiDiagLength + iarsiInputFromDTE[iiInputStartAdd+7];
   
   				CPS(iarsiInputFromDTE[iiInputStartAdd+8],ardiDiagData[0],1);
   				SWPB(ardiDiagData[0],REVERSE,oardiDiagData[0]);
   
   				CPS(iarsiInputFromDTE[iiInputStartAdd+12],ardiDiagData[1],1);
   				SWPB(ardiDiagData[1],REVERSE,oardiDiagData[1]);
   
   				CPS(iarsiInputFromDTE[iiInputStartAdd+16],ardiDiagData[2],1);
   				SWPB(ardiDiagData[2],REVERSE,oardiDiagData[2]);
   
   				CPS(iarsiInputFromDTE[iiInputStartAdd+20],ardiDiagData[3],1);
   				SWPB(ardiDiagData[3],REVERSE,oardiDiagData[3]);
   				iLoopHandlerVar1 := 0;
   
   			ELSE
   				oiDiagLength := oiDiagLength + iarsiInputFromDTE[iiInputStartAdd+3];
   
   				CPS(iarsiInputFromDTE[iiInputStartAdd+6],ardiDiagData[0],1);
   				SWPB(ardiDiagData[0],REVERSE,oardiDiagData[0]);
   
   				CPS(iarsiInputFromDTE[iiInputStartAdd+10],ardiDiagData[1],1);
   				SWPB(ardiDiagData[1],REVERSE,oardiDiagData[1]);
   
   				CPS(iarsiInputFromDTE[iiInputStartAdd+14],ardiDiagData[2],1);
   				SWPB(ardiDiagData[2],REVERSE,oardiDiagData[2]);
   
   				CPS(iarsiInputFromDTE[iiInputStartAdd+18],ardiDiagData[3],1);
   				SWPB(ardiDiagData[3],REVERSE,oardiDiagData[3]);
   				iLoopHandlerVar1 := 0;
   			END_IF;
   
   			IF(oiDiagLength > 0)THEN
   				odiStatus := 16#8000; //Evaluation unit indicates an error; evaluate the diagnostic data in the oardiDiagData output parameter. For the error codes see the device manual
   			ELSE
   				odiStatus := 16#8314;  //Device reported error, but provided no diagonostic codes
   			END_IF;
   
   			iStateMachine_RWH_CMD := 19050;
   		END_IF;
   
   	19050:
   		IF(scDTE102_Handling.Status.DIAG)THEN		// Error in receiving the data from DTE.
   			oxBusy := 1;
   			oxDone := 0;
   			oxError := 0;
   			scDTE102_Handling.ActivateCommand.AO	:= 0;
   			scDTE102_Handling.ActivateCommand.WR	:= 0;
   			scDTE102_Handling.ActivateCommand.RD	:= 0;
   			scDTE102_Handling.ActivateCommand.UR	:= 0;
   			scDTE102_Handling.ActivateCommand.ER	:= 0;
   			scDTE102_Handling.ActivateCommand.DR	:= 1;
   			scDTE102_Handling.ActivateCommand.CM	:= 0;
   			scDTE102_Handling.ActivateCommand.TR	:= NOT(scDTE102_Handling.Status.TA);
   			odiStatus := 16#7402;
   			iStateMachine_RWH_CMD					:= 19000;
   		ELSE
   			iStateMachine_RWH_CMD := 20000;
   		END_IF;
   
   	//Error State According to the error condition, is displayed here
   	20000:
   
   		oxBusy := 0;
   		oxDone := 0;
   		oxError := 1;
   		oiRcvdLength := 0;
   		FOR iLoopHandlerVar1 := 0 TO (iActSizeOfRcvBuf-1) BY 1 DO;
   			oarsiRcvBuf[iLoopHandlerVar1] := 0;
   		END_FOR;
   		iStateMachine_RWH_CMD := 25000;
   
   
   	// Reset all the local and output variable to 0 after Done or Error.
   	25000:
   		IF(oxError)THEN
   			odiStatus := odiStatus;
   		ELSE
   			odiStatus := 16#0000;
   		END_IF;
   		IF(NOT(ixExecute))THEN
   			oxBusy := 0;
   			oxDone := 0;
   			oxError := 0;
   			odiStatus := 16#0000;
   			siActiveFunctionID := 0;
   			iCmdCode := 0;
   			oiRcvdLength := 0;
   			oiDiagLength := 0;
   			ardiDiagData[0] := 0;
   			ardiDiagData[1] := 0;
   			ardiDiagData[2] := 0;
   			ardiDiagData[3] := 0;
   			oardiDiagData[0] := 0;
   			oardiDiagData[1] := 0;
   			oardiDiagData[2] := 0;
   			oardiDiagData[3] := 0;
   			fb_DataLength.Input := 0;
   			INT_TO_BYTE(fb_DataLength);
   			fb_DataAddress.Input := 0;
   			INT_TO_BYTE(fb_DataAddress);
   			FOR iLoopHandlerVar1 :=0 TO (iActSizeOfRcvBuf-1) BY 1 DO;
                               oarsiRcvBuf[iLoopHandlerVar1] := 0;
               END_FOR;
               FOR iLoopHandlerVar2 := (iiInputStartAdd + 2) TO (iiInputStartAdd + iSingleCycleDataExchangeLimitInBytes + 6 -1) BY 1 DO;
                               oarsiOutputToDTE[iLoopHandlerVar2] := 0;
               END_FOR;
   			iLoopHandlerVar1 := 0;
   			iLoopHandlerVar2 := 0;
   
   			iNoCyclesReqToReadWriteCompleteData := 0;
   			iLengthToReadWriteInLastCycle := 0;
   			xMultipleCyclesReq := 0;
   			iBufferOffset := 0;
   			iRcvdLength := 0;
   			iTotalRcvdLength := 0;
   			iActSizeOfInputFromDTE := 0;
   			iActSizeOfOutputToDTE := 0;
   			iActSizeOfRcvBuf := 0;
   			iActSizeOfSendBuf := 0;
   			siActiveModuleID := 0;
   			iActiveInputStartAdd := 0;
   			iActiveOutputStartAdd := 0;
   			iLowerLimitInputStartAdd := 0;
   			iUpperLimitInputStopAdderess := 0;
   			iLowerLimitOutputStartAdd := 0;
   			iUpperLimitOutputStopAdderess := 0;
   
   			iSingleCycleDataExchangeLimitInBytes := 0;
   			fb_SINT_TO_INT.iSINT_var := 0;
   			SINT_TO_INT(fb_SINT_TO_INT,fb_SINT_TO_INT.iSINT_var);
   			iStateMachine_RWH_CMD := 0;
   		END_IF;
   
   	25999: //Wait for ongoing command to complete
   		//If any operation is ongoing, wait for its completion
   		IF(NOT(scDTE102_Handling.Status.TA XOR scDTE102_Handling.ActivateCommand.TR))THEN // Proceed,when TA=TR
   			iStateMachine_RWH_CMD := siActiveFunctionID * ciStateMachineSeparator;
   		END_IF;
   END_CASE;
   
   	IF(iiInputStartAdd >= 0 AND iiInputStartAdd < 496)AND(iiOutputStartAdd >= 0 AND iiOutputStartAdd < 496)THEN
   		// Maping of output bits
   		oarsiOutputToDTE[iiOutputStartAdd].0 := 0;										// Reserve Bit - remain 0 always
   		oarsiOutputToDTE[iiOutputStartAdd].1 := scDTE102_Handling.ActivateCommand.AO;
   		oarsiOutputToDTE[iiOutputStartAdd].2 := scDTE102_Handling.ActivateCommand.WR;
   		oarsiOutputToDTE[iiOutputStartAdd].3 := scDTE102_Handling.ActivateCommand.RD;
   		oarsiOutputToDTE[iiOutputStartAdd].4 := scDTE102_Handling.ActivateCommand.UR;
   		oarsiOutputToDTE[iiOutputStartAdd].5 := scDTE102_Handling.ActivateCommand.ER;
   		oarsiOutputToDTE[iiOutputStartAdd].6 := scDTE102_Handling.ActivateCommand.DR;
   		oarsiOutputToDTE[iiOutputStartAdd].7 := 0;										// Reserve Bit - remain 0 always
   
   		oarsiOutputToDTE[iiOutputStartAdd+1].0 := scDTE102_Handling.ActivateCommand.TR;
   		oarsiOutputToDTE[iiOutputStartAdd+1].1 := 0;										// Reserve Bit - remain 0 always
   		oarsiOutputToDTE[iiOutputStartAdd+1].2 := 0;										// Reserve Bit - remain 0 always
   		oarsiOutputToDTE[iiOutputStartAdd+1].3 := 0;										// Reserve Bit - remain 0 always
   		oarsiOutputToDTE[iiOutputStartAdd+1].4 := 0;										// Reserve Bit - remain 0 always
   		oarsiOutputToDTE[iiOutputStartAdd+1].5 := 0;										// Reserve Bit - remain 0 always
   		oarsiOutputToDTE[iiOutputStartAdd+1].6 := 0;										// Reserve Bit - remain 0 always
   		oarsiOutputToDTE[iiOutputStartAdd+1].7 := scDTE102_Handling.ActivateCommand.CM;
   	END_IF;
   
   
   
   
END_ROUTINE
